LIN {X 0,Y 467.59,Z 100.362,A -85,B 0,C 180,E1 -7607.44,E2 -7607.44} C_VEL
LIN {X 0,Y 467.583,Z 100.361,A -85,B 0,C 180,E1 -7610.855,E2 -7610.855} C_VEL
LIN {X 0,Y 467.561,Z 100.367,A -85,B 0,C 180,E1 -7614.261,E2 -7614.261} C_VEL
LIN {X 0,Y 467.583,Z 100.359,A -85,B 0,C 180,E1 -7617.321,E2 -7617.321} C_VEL
LIN {X 0,Y 467.571,Z 100.367,A -85,B 0,C 180,E1 -7620.667,E2 -7620.667} C_VEL
LIN {X 0,Y 467.632,Z 100.488,A -85,B 0,C 180,E1 -7622.14,E2 -7622.14} C_VEL
LIN {X 0,Y 470.539,Z 113.37,A -85,B 0,C 180,E1 -7624.57,E2 -7624.57} C_VEL
LIN {X 0,Y 471.052,Z 117.501,A -85,B 0,C 180,E1 -7625.307,E2 -7625.307} C_VEL
LIN {X 0,Y 469.859,Z 138.203,A -85,B 0,C 180,E1 -7628.732,E2 -7628.732} C_VEL
LIN {X 0,Y 469.678,Z 141.309,A -85,B 0,C 180,E1 -7629.24,E2 -7629.24} C_VEL
LIN {X 0,Y 473.653,Z 162.605,A -85,B 0,C 180,E1 -7629.783,E2 -7629.783} C_VEL
LIN {X 0,Y 472.479,Z 278.914,A -85,B 0,C 180,E1 -7631.601,E2 -7631.601} C_VEL
LIN {X 0,Y 472.045,Z 293.392,A -85,B 0,C 180,E1 -7631.996,E2 -7631.996} C_VEL
LIN {X 0,Y 471.498,Z 306.65,A -85,B 0,C 180,E1 -7632.524,E2 -7632.524} C_VEL
LIN {X 0,Y 470.833,Z 320.055,A -85,B 0,C 180,E1 -7633.238,E2 -7633.238} C_VEL
LIN {X 0,Y 470.092,Z 333.562,A -85,B 0,C 180,E1 -7634.166,E2 -7634.166} C_VEL
LIN {X 0,Y 469.368,Z 345.002,A -85,B 0,C 180,E1 -7635.142,E2 -7635.142} C_VEL
LIN {X 0,Y 468.685,Z 356.491,A -85,B 0,C 180,E1 -7636.339,E2 -7636.339} C_VEL
LIN {X 0,Y 468.141,Z 365.96,A -85,B 0,C 180,E1 -7637.535,E2 -7637.535} C_VEL
LIN {X 0,Y 467.636,Z 375.295,A -85,B 0,C 180,E1 -7638.953,E2 -7638.953} C_VEL
LIN {X 0,Y 467.209,Z 383.442,A -85,B 0,C 180,E1 -7640.475,E2 -7640.475} C_VEL
LIN {X 0,Y 466.947,Z 389.181,A -85,B 0,C 180,E1 -7641.779,E2 -7641.779} C_VEL
LIN {X 0,Y 466.821,Z 393.865,A -85,B 0,C 180,E1 -7643.082,E2 -7643.082} C_VEL
LIN {X 0,Y 466.723,Z 398.729,A -85,B 0,C 180,E1 -7644.816,E2 -7644.816} C_VEL
LIN {X 0,Y 466.65,Z 402.107,A -85,B 0,C 180,E1 -7646.546,E2 -7646.546} C_VEL
LIN {X 0,Y 466.604,Z 404.094,A -85,B 0,C 180,E1 -7648.274,E2 -7648.274} C_VEL
LIN {X 0,Y 466.598,Z 404.732,A -85,B 0,C 180,E1 -7650,E2 -7650} C_VEL
LIN {X 0,Y 466.604,Z 404.034,A -85,B 0,C 180,E1 -7651.726,E2 -7651.726} C_VEL
LIN {X 0,Y 466.65,Z 401.99,A -85,B 0,C 180,E1 -7653.454,E2 -7653.454} C_VEL
LIN {X 0,Y 466.724,Z 398.543,A -85,B 0,C 180,E1 -7655.184,E2 -7655.184} C_VEL
LIN {X 0,Y 466.82,Z 393.586,A -85,B 0,C 180,E1 -7656.917,E2 -7656.917} C_VEL
LIN {X 0,Y 466.998,Z 386.974,A -85,B 0,C 180,E1 -7658.655,E2 -7658.655} C_VEL
LIN {X 0,Y 467.303,Z 379.612,A -85,B 0,C 180,E1 -7660.178,E2 -7660.178} C_VEL
LIN {X 0,Y 467.801,Z 370.456,A -85,B 0,C 180,E1 -7661.702,E2 -7661.702} C_VEL
LIN {X 0,Y 468.273,Z 360.859,A -85,B 0,C 180,E1 -7663.01,E2 -7663.01} C_VEL
LIN {X 0,Y 468.894,Z 350.221,A -85,B 0,C 180,E1 -7664.207,E2 -7664.207} C_VEL
LIN {X 0,Y 469.535,Z 338.457,A -85,B 0,C 180,E1 -7665.296,E2 -7665.296} C_VEL
LIN {X 0,Y 470.146,Z 326.953,A -85,B 0,C 180,E1 -7666.166,E2 -7666.166} C_VEL
LIN {X 0,Y 470.81,Z 314.697,A -85,B 0,C 180,E1 -7666.91,E2 -7666.91} C_VEL
LIN {X 0,Y 471.344,Z 300.603,A -85,B 0,C 180,E1 -7667.574,E2 -7667.574} C_VEL
LIN {X 0,Y 471.828,Z 287.015,A -85,B 0,C 180,E1 -7668.031,E2 -7668.031} C_VEL
LIN {X 0,Y 472.11,Z 273.417,A -85,B 0,C 180,E1 -7668.329,E2 -7668.329} C_VEL
LIN {X 0,Y 473.107,Z 162.279,A -85,B 0,C 180,E1 -7670.03,E2 -7670.03} C_VEL
LIN {X 0,Y 469.413,Z 141.425,A -85,B 0,C 180,E1 -7670.513,E2 -7670.513} C_VEL
LIN {X 0,Y 470.388,Z 121.167,A -85,B 0,C 180,E1 -7673.791,E2 -7673.791} C_VEL
LIN {X 0,Y 470.519,Z 114.09,A -85,B 0,C 180,E1 -7674.958,E2 -7674.958} C_VEL
LIN {X 0,Y 467.644,Z 100.358,A -85,B 0,C 180,E1 -7677.451,E2 -7677.451} C_VEL
LIN {X 0,Y 467.568,Z 100.367,A -85,B 0,C 180,E1 -7681.045,E2 -7681.045} C_VEL
LIN {X 0,Y 467.588,Z 100.368,A -85,B 0,C 180,E1 -7684.242,E2 -7684.242} C_VEL
LIN {X 0,Y 467.548,Z 100.366,A -85,B 0,C 180,E1 -7687.186,E2 -7687.186} C_VEL
LIN {X 0,Y 467.577,Z 100.366,A -85,B 0,C 180,E1 -7690.264,E2 -7690.264} C_VEL
LIN {X 0,Y 467.586,Z 100.362,A -85,B 0,C 180,E1 -7692.567,E2 -7692.567} C_VEL
LIN {X 0,Y 467.57,Z 100.364,A -85,B 0,C 180,E1 -7695.053,E2 -7695.053} C_VEL
LIN {X 0,Y 467.624,Z 100.361,A -85,B 0,C 180,E1 -7697.444,E2 -7697.444} C_VEL
LIN {X 0,Y 467.559,Z 100.365,A -85,B 0,C 180,E1 -7700.853,E2 -7700.853} C_VEL
LIN {X 0,Y 467.558,Z 100.365,A -85,B 0,C 180,E1 -7704.261,E2 -7704.261} C_VEL
LIN {X 0,Y 467.581,Z 100.369,A -85,B 0,C 180,E1 -7707.321,E2 -7707.321} C_VEL
LIN {X 0,Y 467.569,Z 100.364,A -85,B 0,C 180,E1 -7710.667,E2 -7710.667} C_VEL
LIN {X 0,Y 467.616,Z 100.366,A -85,B 0,C 180,E1 -7713.2,E2 -7713.2} C_VEL
LIN {X 0,Y 467.591,Z 100.362,A -85,B 0,C 180,E1 -7716.468,E2 -7716.468} C_VEL
LIN {X 0,Y 467.621,Z 100.357,A -85,B 0,C 180,E1 -7719.777,E2 -7719.777} C_VEL
LIN {X 0,Y 467.606,Z 100.362,A -85,B 0,C 180,E1 -7722.507,E2 -7722.507} C_VEL
LIN {X 0,Y 467.605,Z 100.362,A -85,B 0,C 180,E1 -7725.197,E2 -7725.197} C_VEL
LIN {X 0,Y 467.655,Z 100.353,A -85,B 0,C 180,E1 -7727.855,E2 -7727.855} C_VEL
LIN {X 0,Y 467.68,Z 100.35,A -85,B 0,C 180,E1 -7731.357,E2 -7731.357} C_VEL
LIN {X 0,Y 467.736,Z 100.344,A -85,B 0,C 180,E1 -7733.963,E2 -7733.963} C_VEL
LIN {X 0,Y 467.858,Z 100.327,A -85,B 0,C 180,E1 -7737.417,E2 -7737.417} C_VEL
LIN {X 0,Y 467.881,Z 100.328,A -85,B 0,C 180,E1 -7740,E2 -7740} C_VEL
LIN {X 0,Y 467.858,Z 100.331,A -85,B 0,C 180,E1 -7742.583,E2 -7742.583} C_VEL
LIN {X 0,Y 467.72,Z 100.352,A -85,B 0,C 180,E1 -7746.038,E2 -7746.038} C_VEL
LIN {X 0,Y 467.681,Z 100.35,A -85,B 0,C 180,E1 -7748.643,E2 -7748.643} C_VEL
LIN {X 0,Y 467.655,Z 100.357,A -85,B 0,C 180,E1 -7752.146,E2 -7752.146} C_VEL
LIN {X 0,Y 467.638,Z 100.361,A -85,B 0,C 180,E1 -7755.695,E2 -7755.695} C_VEL
LIN {X 0,Y 467.621,Z 100.36,A -85,B 0,C 180,E1 -7759.308,E2 -7759.308} C_VEL
LIN {X 0,Y 467.534,Z 100.37,A -85,B 0,C 180,E1 -7762.074,E2 -7762.074} C_VEL
LIN {X 0,Y 467.585,Z 100.363,A -85,B 0,C 180,E1 -7764.889,E2 -7764.889} C_VEL
LIN {X 0,Y 467.619,Z 100.36,A -85,B 0,C 180,E1 -7767.769,E2 -7767.769} C_VEL
LIN {X 0,Y 467.567,Z 100.368,A -85,B 0,C 180,E1 -7771.045,E2 -7771.045} C_VEL
LIN {X 0,Y 467.577,Z 100.362,A -85,B 0,C 180,E1 -7774.24,E2 -7774.24} C_VEL
LIN {X 0,Y 467.547,Z 100.372,A -85,B 0,C 180,E1 -7777.187,E2 -7777.187} C_VEL
LIN {X 0,Y 467.574,Z 100.363,A -85,B 0,C 180,E1 -7780.265,E2 -7780.265} C_VEL
LIN {X 0,Y 467.587,Z 100.365,A -85,B 0,C 180,E1 -7782.567,E2 -7782.567} C_VEL
LIN {X 0,Y 467.566,Z 100.368,A -85,B 0,C 180,E1 -7785.053,E2 -7785.053} C_VEL
LIN {X 0,Y 467.574,Z 100.369,A -85,B 0,C 180,E1 -7788.597,E2 -7788.597} C_VEL
LIN {X 0,Y 467.563,Z 100.365,A -85,B 0,C 180,E1 -7791.956,E2 -7791.956} C_VEL
LIN {X 0,Y 467.564,Z 100.365,A -85,B 0,C 180,E1 -7795.168,E2 -7795.168} C_VEL
LIN {X 0,Y 467.585,Z 100.368,A -85,B 0,C 180,E1 -7798.26,E2 -7798.26} C_VEL
LIN {X 0,Y 467.556,Z 100.365,A -85,B 0,C 180,E1 -7801.249,E2 -7801.249} C_VEL
LIN {X 0,Y 467.581,Z 100.369,A -85,B 0,C 180,E1 -7804.159,E2 -7804.159} C_VEL
LIN {X 0,Y 467.578,Z 100.362,A -85,B 0,C 180,E1 -7806.996,E2 -7806.996} C_VEL
LIN {X 0,Y 467.611,Z 100.363,A -85,B 0,C 180,E1 -7810.375,E2 -7810.375} C_VEL
LIN {X 0,Y 467.649,Z 100.469,A -85,B 0,C 180,E1 -7811.446,E2 -7811.446} C_VEL
LIN {X 0,Y 469.89,Z 112.337,A -85,B 0,C 180,E1 -7813.801,E2 -7813.801} C_VEL
LIN {X 0,Y 469.308,Z 114.722,A -85,B 0,C 180,E1 -7814.217,E2 -7814.217} C_VEL
LIN {X 0,Y 467.724,Z 117.234,A -85,B 0,C 180,E1 -7814.59,E2 -7814.59} C_VEL
LIN {X 0,Y 465.302,Z 120.97,A -85,B 0,C 180,E1 -7815.008,E2 -7815.008} C_VEL
LIN {X 0,Y 463.889,Z 124.864,A -85,B 0,C 180,E1 -7815.289,E2 -7815.289} C_VEL
LIN {X 0,Y 463.925,Z 127.986,A -85,B 0,C 180,E1 -7815.416,E2 -7815.416} C_VEL
LIN {X 0,Y 466.531,Z 140.838,A -85,B 0,C 180,E1 -7815.733,E2 -7815.733} C_VEL
LIN {X 0,Y 465.376,Z 258.301,A -85,B 0,C 180,E1 -7817.573,E2 -7817.573} C_VEL
LIN {X 0,Y 465.029,Z 272.977,A -85,B 0,C 180,E1 -7817.979,E2 -7817.979} C_VEL
LIN {X 0,Y 464.568,Z 286.896,A -85,B 0,C 180,E1 -7818.548,E2 -7818.548} C_VEL
LIN {X 0,Y 463.909,Z 300.717,A -85,B 0,C 180,E1 -7819.305,E2 -7819.305} C_VEL
LIN {X 0,Y 463.223,Z 313.085,A -85,B 0,C 180,E1 -7820.173,E2 -7820.173} C_VEL
LIN {X 0,Y 462.552,Z 325.536,A -85,B 0,C 180,E1 -7821.261,E2 -7821.261} C_VEL
LIN {X 0,Y 461.968,Z 335.732,A -85,B 0,C 180,E1 -7822.351,E2 -7822.351} C_VEL
LIN {X 0,Y 461.293,Z 345.908,A -85,B 0,C 180,E1 -7823.659,E2 -7823.659} C_VEL
LIN {X 0,Y 460.791,Z 354.325,A -85,B 0,C 180,E1 -7824.969,E2 -7824.969} C_VEL
LIN {X 0,Y 460.197,Z 362.395,A -85,B 0,C 180,E1 -7826.498,E2 -7826.498} C_VEL
LIN {X 0,Y 460.018,Z 368.058,A -85,B 0,C 180,E1 -7827.811,E2 -7827.811} C_VEL
LIN {X 0,Y 459.705,Z 372.702,A -85,B 0,C 180,E1 -7829.124,E2 -7829.124} C_VEL
LIN {X 0,Y 459.615,Z 377.518,A -85,B 0,C 180,E1 -7830.876,E2 -7830.876} C_VEL
LIN {X 0,Y 459.601,Z 380.867,A -85,B 0,C 180,E1 -7832.629,E2 -7832.629} C_VEL
LIN {X 0,Y 459.521,Z 382.844,A -85,B 0,C 180,E1 -7834.386,E2 -7834.386} C_VEL
LIN {X 0,Y 459.592,Z 383.48,A -85,B 0,C 180,E1 -7836.145,E2 -7836.145} C_VEL
LIN {X 0,Y 459.522,Z 382.783,A -85,B 0,C 180,E1 -7837.912,E2 -7837.912} C_VEL
LIN {X 0,Y 459.505,Z 380.734,A -85,B 0,C 180,E1 -7839.686,E2 -7839.686} C_VEL
LIN {X 0,Y 459.744,Z 377.272,A -85,B 0,C 180,E1 -7841.463,E2 -7841.463} C_VEL
LIN {X 0,Y 459.91,Z 372.284,A -85,B 0,C 180,E1 -7843.251,E2 -7843.251} C_VEL
LIN {X 0,Y 460.144,Z 367.43,A -85,B 0,C 180,E1 -7844.597,E2 -7844.597} C_VEL
LIN {X 0,Y 460.56,Z 360.387,A -85,B 0,C 180,E1 -7846.17,E2 -7846.17} C_VEL
LIN {X 0,Y 461.093,Z 351.616,A -85,B 0,C 180,E1 -7847.749,E2 -7847.749} C_VEL
LIN {X 0,Y 461.759,Z 341.549,A -85,B 0,C 180,E1 -7849.219,E2 -7849.219} C_VEL
LIN {X 0,Y 462.573,Z 330.076,A -85,B 0,C 180,E1 -7850.57,E2 -7850.57} C_VEL
LIN {X 0,Y 463.306,Z 318.29,A -85,B 0,C 180,E1 -7851.7,E2 -7851.7} C_VEL
LIN {X 0,Y 464.113,Z 305.504,A -85,B 0,C 180,E1 -7852.688,E2 -7852.688} C_VEL
LIN {X 0,Y 464.802,Z 292.175,A -85,B 0,C 180,E1 -7853.503,E2 -7853.503} C_VEL
LIN {X 0,Y 465.368,Z 278.873,A -85,B 0,C 180,E1 -7854.123,E2 -7854.123} C_VEL
LIN {X 0,Y 465.805,Z 265.448,A -85,B 0,C 180,E1 -7854.574,E2 -7854.574} C_VEL
LIN {X 0,Y 466.093,Z 250.619,A -85,B 0,C 180,E1 -7854.884,E2 -7854.884} C_VEL
LIN {X 0,Y 467.2,Z 140.6,A -85,B 0,C 180,E1 -7856.616,E2 -7856.616} C_VEL
LIN {X 0,Y 463.098,Z 122.09,A -85,B 0,C 180,E1 -7857.144,E2 -7857.144} C_VEL
LIN {X 0,Y 463.355,Z 115.546,A -85,B 0,C 180,E1 -7858.391,E2 -7858.391} C_VEL
LIN {X 0,Y 461.497,Z 105.781,A -85,B 0,C 180,E1 -7860.421,E2 -7860.421} C_VEL
LIN {X 0,Y 460.521,Z 101.248,A -85,B 0,C 180,E1 -7861.407,E2 -7861.407} C_VEL
LIN {X 0,Y 460.509,Z 101.246,A -85,B 0,C 180,E1 -7864.501,E2 -7864.501} C_VEL
LIN {X 0,Y 460.482,Z 101.25,A -85,B 0,C 180,E1 -7867.625,E2 -7867.625} C_VEL
LIN {X 0,Y 460.5,Z 101.247,A -85,B 0,C 180,E1 -7871.015,E2 -7871.015} C_VEL
LIN {X 0,Y 460.51,Z 101.244,A -85,B 0,C 180,E1 -7874.589,E2 -7874.589} C_VEL
LIN {X 0,Y 460.476,Z 101.252,A -85,B 0,C 180,E1 -7877.813,E2 -7877.813} C_VEL
LIN {X 0,Y 460.511,Z 101.236,A -85,B 0,C 180,E1 -7880.135,E2 -7880.135} C_VEL
LIN {X 0,Y 460.466,Z 101.252,A -85,B 0,C 180,E1 -7883.469,E2 -7883.469} C_VEL
LIN {X 0,Y 460.52,Z 101.244,A -85,B 0,C 180,E1 -7886.674,E2 -7886.674} C_VEL
LIN {X 0,Y 460.505,Z 101.242,A -85,B 0,C 180,E1 -7889.759,E2 -7889.759} C_VEL
LIN {X 0,Y 460.512,Z 101.249,A -85,B 0,C 180,E1 -7892.752,E2 -7892.752} C_VEL
LIN {X 0,Y 460.517,Z 101.243,A -85,B 0,C 180,E1 -7895.666,E2 -7895.666} C_VEL
LIN {X 0,Y 460.523,Z 101.243,A -85,B 0,C 180,E1 -7898.578,E2 -7898.578} C_VEL
LIN {X 0,Y 460.586,Z 101.23,A -85,B 0,C 180,E1 -7901.311,E2 -7901.311} C_VEL
LIN {X 0,Y 460.606,Z 101.234,A -85,B 0,C 180,E1 -7904.059,E2 -7904.059} C_VEL
LIN {X 0,Y 460.61,Z 101.23,A -85,B 0,C 180,E1 -7907.666,E2 -7907.666} C_VEL
LIN {X 0,Y 460.62,Z 101.223,A -85,B 0,C 180,E1 -7911.224,E2 -7911.224} C_VEL
LIN {X 0,Y 460.685,Z 101.226,A -85,B 0,C 180,E1 -7913.87,E2 -7913.87} C_VEL
LIN {X 0,Y 460.792,Z 101.206,A -85,B 0,C 180,E1 -7917.377,E2 -7917.377} C_VEL
LIN {X 0,Y 460.852,Z 101.203,A -85,B 0,C 180,E1 -7920,E2 -7920} C_VEL
LIN {X 0,Y 460.793,Z 101.208,A -85,B 0,C 180,E1 -7922.622,E2 -7922.622} C_VEL
LIN {X 0,Y 460.678,Z 101.22,A -85,B 0,C 180,E1 -7926.13,E2 -7926.13} C_VEL
LIN {X 0,Y 460.621,Z 101.23,A -85,B 0,C 180,E1 -7928.776,E2 -7928.776} C_VEL
LIN {X 0,Y 460.614,Z 101.228,A -85,B 0,C 180,E1 -7932.445,E2 -7932.445} C_VEL
LIN {X 0,Y 460.601,Z 101.226,A -85,B 0,C 180,E1 -7935.997,E2 -7935.997} C_VEL
LIN {X 0,Y 460.572,Z 101.238,A -85,B 0,C 180,E1 -7938.902,E2 -7938.902} C_VEL
LIN {X 0,Y 460.517,Z 101.244,A -85,B 0,C 180,E1 -7941.485,E2 -7941.485} C_VEL
LIN {X 0,Y 460.542,Z 101.237,A -85,B 0,C 180,E1 -7944.332,E2 -7944.332} C_VEL
LIN {X 0,Y 460.574,Z 101.238,A -85,B 0,C 180,E1 -7947.244,E2 -7947.244} C_VEL
LIN {X 0,Y 460.512,Z 101.243,A -85,B 0,C 180,E1 -7950.24,E2 -7950.24} C_VEL
LIN {X 0,Y 460.53,Z 101.243,A -85,B 0,C 180,E1 -7953.325,E2 -7953.325} C_VEL
LIN {X 0,Y 460.477,Z 101.252,A -85,B 0,C 180,E1 -7956.529,E2 -7956.529} C_VEL
LIN {X 0,Y 460.526,Z 101.234,A -85,B 0,C 180,E1 -7959.863,E2 -7959.863} C_VEL
LIN {X 0,Y 460.513,Z 101.244,A -85,B 0,C 180,E1 -7962.9,E2 -7962.9} C_VEL
LIN {X 0,Y 460.51,Z 101.243,A -85,B 0,C 180,E1 -7965.831,E2 -7965.831} C_VEL
LIN {X 0,Y 460.532,Z 101.241,A -85,B 0,C 180,E1 -7968.989,E2 -7968.989} C_VEL
LIN {X 0,Y 460.527,Z 101.24,A -85,B 0,C 180,E1 -7971.267,E2 -7971.267} C_VEL
LIN {X 0,Y 460.511,Z 101.243,A -85,B 0,C 180,E1 -7974.554,E2 -7974.554} C_VEL
LIN {X 0,Y 460.532,Z 101.24,A -85,B 0,C 180,E1 -7977.716,E2 -7977.716} C_VEL
LIN {X 0,Y 460.541,Z 101.243,A -85,B 0,C 180,E1 -7980.769,E2 -7980.769} C_VEL
LIN {X 0,Y 460.609,Z 101.434,A -85,B 0,C 180,E1 -7981.838,E2 -7981.838} C_VEL
LIN {X 0,Y 463.648,Z 114.783,A -85,B 0,C 180,E1 -7984.405,E2 -7984.405} C_VEL
LIN {X 0,Y 464.173,Z 119.706,A -85,B 0,C 180,E1 -7985.293,E2 -7985.293} C_VEL
LIN {X 0,Y 462.942,Z 139.583,A -85,B 0,C 180,E1 -7988.632,E2 -7988.632} C_VEL
LIN {X 0,Y 462.848,Z 141.135,A -85,B 0,C 180,E1 -7988.891,E2 -7988.891} C_VEL
LIN {X 0,Y 467.042,Z 163.344,A -85,B 0,C 180,E1 -7989.473,E2 -7989.473} C_VEL
LIN {X 0,Y 465.804,Z 278.587,A -85,B 0,C 180,E1 -7991.3,E2 -7991.3} C_VEL
LIN {X 0,Y 465.347,Z 293.36,A -85,B 0,C 180,E1 -7991.708,E2 -7991.708} C_VEL
LIN {X 0,Y 464.723,Z 307.37,A -85,B 0,C 180,E1 -7992.281,E2 -7992.281} C_VEL
LIN {X 0,Y 464.039,Z 320.484,A -85,B 0,C 180,E1 -7993,E2 -7993} C_VEL
LIN {X 0,Y 463.268,Z 333.695,A -85,B 0,C 180,E1 -7993.927,E2 -7993.927} C_VEL
LIN {X 0,Y 462.423,Z 346.25,A -85,B 0,C 180,E1 -7995.027,E2 -7995.027} C_VEL
LIN {X 0,Y 461.761,Z 356.524,A -85,B 0,C 180,E1 -7996.13,E2 -7996.13} C_VEL
LIN {X 0,Y 461.131,Z 366.58,A -85,B 0,C 180,E1 -7997.429,E2 -7997.429} C_VEL
LIN {X 0,Y 460.639,Z 375.254,A -85,B 0,C 180,E1 -7998.783,E2 -7998.783} C_VEL
LIN {X 0,Y 460.175,Z 383.372,A -85,B 0,C 180,E1 -8000.329,E2 -8000.329} C_VEL
LIN {X 0,Y 459.896,Z 389.099,A -85,B 0,C 180,E1 -8001.652,E2 -8001.652} C_VEL
LIN {X 0,Y 459.731,Z 393.764,A -85,B 0,C 180,E1 -8002.975,E2 -8002.975} C_VEL
LIN {X 0,Y 459.635,Z 398.612,A -85,B 0,C 180,E1 -8004.736,E2 -8004.736} C_VEL
LIN {X 0,Y 459.546,Z 401.974,A -85,B 0,C 180,E1 -8006.493,E2 -8006.493} C_VEL
LIN {X 0,Y 459.517,Z 403.944,A -85,B 0,C 180,E1 -8008.247,E2 -8008.247} C_VEL
LIN {X 0,Y 459.501,Z 404.567,A -85,B 0,C 180,E1 -8010,E2 -8010} C_VEL
LIN {X 0,Y 459.517,Z 403.855,A -85,B 0,C 180,E1 -8011.753,E2 -8011.753} C_VEL
LIN {X 0,Y 459.547,Z 401.796,A -85,B 0,C 180,E1 -8013.507,E2 -8013.507} C_VEL
LIN {X 0,Y 459.632,Z 398.333,A -85,B 0,C 180,E1 -8015.264,E2 -8015.264} C_VEL
LIN {X 0,Y 459.731,Z 393.359,A -85,B 0,C 180,E1 -8017.025,E2 -8017.025} C_VEL
LIN {X 0,Y 459.941,Z 386.728,A -85,B 0,C 180,E1 -8018.789,E2 -8018.789} C_VEL
LIN {X 0,Y 460.276,Z 379.344,A -85,B 0,C 180,E1 -8020.335,E2 -8020.335} C_VEL
LIN {X 0,Y 460.764,Z 370.149,A -85,B 0,C 180,E1 -8021.883,E2 -8021.883} C_VEL
LIN {X 0,Y 461.304,Z 360.521,A -85,B 0,C 180,E1 -8023.21,E2 -8023.21} C_VEL
LIN {X 0,Y 461.974,Z 349.845,A -85,B 0,C 180,E1 -8024.425,E2 -8024.425} C_VEL
LIN {X 0,Y 462.653,Z 338.031,A -85,B 0,C 180,E1 -8025.529,E2 -8025.529} C_VEL
LIN {X 0,Y 463.297,Z 326.464,A -85,B 0,C 180,E1 -8026.411,E2 -8026.411} C_VEL
LIN {X 0,Y 464.053,Z 313.041,A -85,B 0,C 180,E1 -8027.225,E2 -8027.225} C_VEL
LIN {X 0,Y 464.522,Z 299.889,A -85,B 0,C 180,E1 -8027.841,E2 -8027.841} C_VEL
LIN {X 0,Y 465.058,Z 286.076,A -85,B 0,C 180,E1 -8028.303,E2 -8028.303} C_VEL
LIN {X 0,Y 465.356,Z 271.908,A -85,B 0,C 180,E1 -8028.605,E2 -8028.605} C_VEL
LIN {X 0,Y 466.361,Z 163.164,A -85,B 0,C 180,E1 -8030.291,E2 -8030.291} C_VEL
LIN {X 0,Y 462.503,Z 141.199,A -85,B 0,C 180,E1 -8030.817,E2 -8030.817} C_VEL
LIN {X 0,Y 463.491,Z 122.252,A -85,B 0,C 180,E1 -8033.929,E2 -8033.929} C_VEL
LIN {X 0,Y 463.553,Z 115.172,A -85,B 0,C 180,E1 -8035.12,E2 -8035.12} C_VEL
LIN {X 0,Y 460.595,Z 101.236,A -85,B 0,C 180,E1 -8037.702,E2 -8037.702} C_VEL
LIN {X 0,Y 460.521,Z 101.245,A -85,B 0,C 180,E1 -8041.283,E2 -8041.283} C_VEL
LIN {X 0,Y 460.532,Z 101.243,A -85,B 0,C 180,E1 -8044.505,E2 -8044.505} C_VEL
LIN {X 0,Y 460.501,Z 101.246,A -85,B 0,C 180,E1 -8047.623,E2 -8047.623} C_VEL
LIN {X 0,Y 460.541,Z 101.242,A -85,B 0,C 180,E1 -8050.269,E2 -8050.269} C_VEL
LIN {X 0,Y 460.499,Z 101.246,A -85,B 0,C 180,E1 -8053.375,E2 -8053.375} C_VEL
LIN {X 0,Y 460.524,Z 101.241,A -85,B 0,C 180,E1 -8056.627,E2 -8056.627} C_VEL
LIN {X 0,Y 460.539,Z 101.246,A -85,B 0,C 180,E1 -8059.731,E2 -8059.731} C_VEL
LIN {X 0,Y 460.498,Z 101.244,A -85,B 0,C 180,E1 -8062.524,E2 -8062.524} C_VEL
LIN {X 0,Y 460.545,Z 101.244,A -85,B 0,C 180,E1 -8065.624,E2 -8065.624} C_VEL
LIN {X 0,Y 460.536,Z 101.241,A -85,B 0,C 180,E1 -8068.744,E2 -8068.744} C_VEL
LIN {X 0,Y 460.58,Z 101.234,A -85,B 0,C 180,E1 -8072.254,E2 -8072.254} C_VEL
LIN {X 0,Y 460.557,Z 101.239,A -85,B 0,C 180,E1 -8074.705,E2 -8074.705} C_VEL
LIN {X 0,Y 460.509,Z 101.244,A -85,B 0,C 180,E1 -8077.571,E2 -8077.571} C_VEL
LIN {X 0,Y 460.567,Z 101.237,A -85,B 0,C 180,E1 -8080.385,E2 -8080.385} C_VEL
LIN {X 0,Y 460.563,Z 101.24,A -85,B 0,C 180,E1 -8083.146,E2 -8083.146} C_VEL
LIN {X 0,Y 460.554,Z 101.237,A -85,B 0,C 180,E1 -8085.868,E2 -8085.868} C_VEL
LIN {X 0,Y 460.61,Z 101.236,A -85,B 0,C 180,E1 -8088.559,E2 -8088.559} C_VEL
LIN {X 0,Y 460.694,Z 101.222,A -85,B 0,C 180,E1 -8092.109,E2 -8092.109} C_VEL
LIN {X 0,Y 460.694,Z 101.224,A -85,B 0,C 180,E1 -8094.748,E2 -8094.748} C_VEL
LIN {X 0,Y 460.799,Z 101.207,A -85,B 0,C 180,E1 -8097.378,E2 -8097.378} C_VEL
LIN {X 0,Y 460.852,Z 101.204,A -85,B 0,C 180,E1 -8100,E2 -8100} C_VEL
LIN {X 0,Y 460.799,Z 101.209,A -85,B 0,C 180,E1 -8102.623,E2 -8102.623} C_VEL
LIN {X 0,Y 460.684,Z 101.229,A -85,B 0,C 180,E1 -8106.13,E2 -8106.13} C_VEL
LIN {X 0,Y 460.628,Z 101.228,A -85,B 0,C 180,E1 -8108.776,E2 -8108.776} C_VEL
LIN {X 0,Y 460.613,Z 101.231,A -85,B 0,C 180,E1 -8112.445,E2 -8112.445} C_VEL
LIN {X 0,Y 460.6,Z 101.236,A -85,B 0,C 180,E1 -8115.998,E2 -8115.998} C_VEL
LIN {X 0,Y 460.567,Z 101.243,A -85,B 0,C 180,E1 -8119.616,E2 -8119.616} C_VEL
LIN {X 0,Y 460.51,Z 101.243,A -85,B 0,C 180,E1 -8122.429,E2 -8122.429} C_VEL
LIN {X 0,Y 460.552,Z 101.241,A -85,B 0,C 180,E1 -8125.798,E2 -8125.798} C_VEL
LIN {X 0,Y 460.551,Z 101.238,A -85,B 0,C 180,E1 -8128.233,E2 -8128.233} C_VEL
LIN {X 0,Y 460.52,Z 101.249,A -85,B 0,C 180,E1 -8131.283,E2 -8131.283} C_VEL
LIN {X 0,Y 460.523,Z 101.242,A -85,B 0,C 180,E1 -8134.504,E2 -8134.504} C_VEL
LIN {X 0,Y 460.501,Z 101.245,A -85,B 0,C 180,E1 -8137.624,E2 -8137.624} C_VEL
LIN {X 0,Y 460.539,Z 101.24,A -85,B 0,C 180,E1 -8140.269,E2 -8140.269} C_VEL
LIN {X 0,Y 460.497,Z 101.246,A -85,B 0,C 180,E1 -8143.376,E2 -8143.376} C_VEL
LIN {X 0,Y 460.509,Z 101.249,A -85,B 0,C 180,E1 -8146.626,E2 -8146.626} C_VEL
LIN {X 0,Y 460.536,Z 101.239,A -85,B 0,C 180,E1 -8149.732,E2 -8149.732} C_VEL
LIN {X 0,Y 460.498,Z 101.252,A -85,B 0,C 180,E1 -8152.525,E2 -8152.525} C_VEL
LIN {X 0,Y 460.547,Z 101.238,A -85,B 0,C 180,E1 -8155.624,E2 -8155.624} C_VEL
LIN {X 0,Y 460.539,Z 101.242,A -85,B 0,C 180,E1 -8158.745,E2 -8158.745} C_VEL
LIN {X 0,Y 460.552,Z 101.245,A -85,B 0,C 180,E1 -8162.262,E2 -8162.262} C_VEL
LIN {X 0,Y 460.536,Z 101.241,A -85,B 0,C 180,E1 -8164.704,E2 -8164.704} C_VEL
LIN {X 0,Y 460.513,Z 101.244,A -85,B 0,C 180,E1 -8167.572,E2 -8167.572} C_VEL
LIN {X 0,Y 460.57,Z 101.242,A -85,B 0,C 180,E1 -8170.385,E2 -8170.385} C_VEL
LIN {X 0,Y 460.589,Z 101.323,A -85,B 0,C 180,E1 -8171.215,E2 -8171.215} C_VEL
LIN {X 0,Y 462.976,Z 113.738,A -85,B 0,C 180,E1 -8173.717,E2 -8173.717} C_VEL
LIN {X 0,Y 462.7,Z 122.021,A -85,B 0,C 180,E1 -8175.261,E2 -8175.261} C_VEL
LIN {X 0,Y 463.925,Z 127.986,A -85,B 0,C 180,E1 -8175.416,E2 -8175.416} C_VEL
LIN {X 0,Y 464.359,Z 133.792,A -85,B 0,C 180,E1 -8175.528,E2 -8175.528} C_VEL
LIN {X 0,Y 463.604,Z 139.673,A -85,B 0,C 180,E1 -8175.59,E2 -8175.59} C_VEL
LIN {X 0,Y 460.035,Z 155.401,A -85,B 0,C 180,E1 -8175.693,E2 -8175.693} C_VEL
LIN {X 0,Y 459.698,Z 159.403,A -85,B 0,C 180,E1 -8175.743,E2 -8175.743} C_VEL
LIN {X 0,Y 458.593,Z 259.062,A -85,B 0,C 180,E1 -8177.33,E2 -8177.33} C_VEL
LIN {X 0,Y 458.233,Z 273.507,A -85,B 0,C 180,E1 -8177.742,E2 -8177.742} C_VEL
LIN {X 0,Y 457.75,Z 287.335,A -85,B 0,C 180,E1 -8178.319,E2 -8178.319} C_VEL
LIN {X 0,Y 457.109,Z 300.226,A -85,B 0,C 180,E1 -8179.032,E2 -8179.032} C_VEL
LIN {X 0,Y 456.393,Z 312.723,A -85,B 0,C 180,E1 -8179.912,E2 -8179.912} C_VEL
LIN {X 0,Y 455.678,Z 325.021,A -85,B 0,C 180,E1 -8180.992,E2 -8180.992} C_VEL
LIN {X 0,Y 454.993,Z 336.5,A -85,B 0,C 180,E1 -8182.233,E2 -8182.233} C_VEL
LIN {X 0,Y 454.273,Z 346.547,A -85,B 0,C 180,E1 -8183.56,E2 -8183.56} C_VEL
LIN {X 0,Y 453.763,Z 354.889,A -85,B 0,C 180,E1 -8184.891,E2 -8184.891} C_VEL
LIN {X 0,Y 453.153,Z 362.879,A -85,B 0,C 180,E1 -8186.443,E2 -8186.443} C_VEL
LIN {X 0,Y 452.931,Z 368.508,A -85,B 0,C 180,E1 -8187.777,E2 -8187.777} C_VEL
LIN {X 0,Y 452.661,Z 374.429,A -85,B 0,C 180,E1 -8189.555,E2 -8189.555} C_VEL
LIN {X 0,Y 452.546,Z 377.853,A -85,B 0,C 180,E1 -8190.89,E2 -8190.89} C_VEL
LIN {X 0,Y 452.522,Z 381.145,A -85,B 0,C 180,E1 -8192.671,E2 -8192.671} C_VEL
LIN {X 0,Y 452.438,Z 383.057,A -85,B 0,C 180,E1 -8194.455,E2 -8194.455} C_VEL
LIN {X 0,Y 452.516,Z 383.623,A -85,B 0,C 180,E1 -8196.287,E2 -8196.287} C_VEL
LIN {X 0,Y 452.439,Z 382.881,A -85,B 0,C 180,E1 -8198.037,E2 -8198.037} C_VEL
LIN {X 0,Y 452.429,Z 380.778,A -85,B 0,C 180,E1 -8199.839,E2 -8199.839} C_VEL
LIN {X 0,Y 452.674,Z 377.262,A -85,B 0,C 180,E1 -8201.644,E2 -8201.644} C_VEL
LIN {X 0,Y 452.866,Z 372.216,A -85,B 0,C 180,E1 -8203.461,E2 -8203.461} C_VEL
LIN {X 0,Y 453.127,Z 367.299,A -85,B 0,C 180,E1 -8204.828,E2 -8204.828} C_VEL
LIN {X 0,Y 453.594,Z 360.188,A -85,B 0,C 180,E1 -8206.425,E2 -8206.425} C_VEL
LIN {X 0,Y 454.076,Z 352.712,A -85,B 0,C 180,E1 -8207.799,E2 -8207.799} C_VEL
LIN {X 0,Y 454.695,Z 343.678,A -85,B 0,C 180,E1 -8209.176,E2 -8209.176} C_VEL
LIN {X 0,Y 455.386,Z 334.686,A -85,B 0,C 180,E1 -8210.319,E2 -8210.319} C_VEL
LIN {X 0,Y 456.12,Z 323.897,A -85,B 0,C 180,E1 -8211.466,E2 -8211.466} C_VEL
LIN {X 0,Y 456.98,Z 311.373,A -85,B 0,C 180,E1 -8212.549,E2 -8212.549} C_VEL
LIN {X 0,Y 457.756,Z 298.993,A -85,B 0,C 180,E1 -8213.407,E2 -8213.407} C_VEL
LIN {X 0,Y 458.479,Z 285.304,A -85,B 0,C 180,E1 -8214.148,E2 -8214.148} C_VEL
LIN {X 0,Y 458.96,Z 271.706,A -85,B 0,C 180,E1 -8214.693,E2 -8214.693} C_VEL
LIN {X 0,Y 459.354,Z 257.984,A -85,B 0,C 180,E1 -8215.063,E2 -8215.063} C_VEL
LIN {X 0,Y 460.667,Z 141.91,A -85,B 0,C 180,E1 -8216.93,E2 -8216.93} C_VEL
LIN {X 0,Y 456.293,Z 122.254,A -85,B 0,C 180,E1 -8217.506,E2 -8217.506} C_VEL
LIN {X 0,Y 456.401,Z 116.481,A -85,B 0,C 180,E1 -8218.63,E2 -8218.63} C_VEL
LIN {X 0,Y 454.224,Z 105.584,A -85,B 0,C 180,E1 -8220.947,E2 -8220.947} C_VEL
LIN {X 0,Y 453.464,Z 102.128,A -85,B 0,C 180,E1 -8221.71,E2 -8221.71} C_VEL
LIN {X 0,Y 453.467,Z 102.122,A -85,B 0,C 180,E1 -8224.99,E2 -8224.99} C_VEL
LIN {X 0,Y 453.441,Z 102.128,A -85,B 0,C 180,E1 -8228.314,E2 -8228.314} C_VEL
LIN {X 0,Y 453.465,Z 102.123,A -85,B 0,C 180,E1 -8230.612,E2 -8230.612} C_VEL
LIN {X 0,Y 453.48,Z 102.12,A -85,B 0,C 180,E1 -8234.528,E2 -8234.528} C_VEL
LIN {X 0,Y 453.437,Z 102.127,A -85,B 0,C 180,E1 -8238.071,E2 -8238.071} C_VEL
LIN {X 0,Y 453.439,Z 102.117,A -85,B 0,C 180,E1 -8240.802,E2 -8240.802} C_VEL
LIN {X 0,Y 453.448,Z 102.122,A -85,B 0,C 180,E1 -8243.916,E2 -8243.916} C_VEL
LIN {X 0,Y 453.479,Z 102.123,A -85,B 0,C 180,E1 -8247.151,E2 -8247.151} C_VEL
LIN {X 0,Y 453.463,Z 102.119,A -85,B 0,C 180,E1 -8250.267,E2 -8250.267} C_VEL
LIN {X 0,Y 453.453,Z 102.122,A -85,B 0,C 180,E1 -8253.29,E2 -8253.29} C_VEL
LIN {X 0,Y 453.493,Z 102.119,A -85,B 0,C 180,E1 -8256.238,E2 -8256.238} C_VEL
LIN {X 0,Y 453.483,Z 102.122,A -85,B 0,C 180,E1 -8259.117,E2 -8259.117} C_VEL
LIN {X 0,Y 453.502,Z 102.113,A -85,B 0,C 180,E1 -8261.944,E2 -8261.944} C_VEL
LIN {X 0,Y 453.536,Z 102.115,A -85,B 0,C 180,E1 -8264.726,E2 -8264.726} C_VEL
LIN {X 0,Y 453.56,Z 102.115,A -85,B 0,C 180,E1 -8268.379,E2 -8268.379} C_VEL
LIN {X 0,Y 453.586,Z 102.1,A -85,B 0,C 180,E1 -8271.086,E2 -8271.086} C_VEL
LIN {X 0,Y 453.651,Z 102.101,A -85,B 0,C 180,E1 -8273.774,E2 -8273.774} C_VEL
LIN {X 0,Y 453.736,Z 102.085,A -85,B 0,C 180,E1 -8277.336,E2 -8277.336} C_VEL
LIN {X 0,Y 453.822,Z 102.078,A -85,B 0,C 180,E1 -8280,E2 -8280} C_VEL
LIN {X 0,Y 453.737,Z 102.086,A -85,B 0,C 180,E1 -8282.663,E2 -8282.663} C_VEL
LIN {X 0,Y 453.645,Z 102.095,A -85,B 0,C 180,E1 -8286.226,E2 -8286.226} C_VEL
LIN {X 0,Y 453.586,Z 102.107,A -85,B 0,C 180,E1 -8288.913,E2 -8288.913} C_VEL
LIN {X 0,Y 453.564,Z 102.106,A -85,B 0,C 180,E1 -8292.529,E2 -8292.529} C_VEL
LIN {X 0,Y 453.546,Z 102.104,A -85,B 0,C 180,E1 -8296.196,E2 -8296.196} C_VEL
LIN {X 0,Y 453.521,Z 102.118,A -85,B 0,C 180,E1 -8299.041,E2 -8299.041} C_VEL
LIN {X 0,Y 453.477,Z 102.118,A -85,B 0,C 180,E1 -8301.836,E2 -8301.836} C_VEL
LIN {X 0,Y 453.514,Z 102.116,A -85,B 0,C 180,E1 -8304.734,E2 -8304.734} C_VEL
LIN {X 0,Y 453.533,Z 102.111,A -85,B 0,C 180,E1 -8307.96,E2 -8307.96} C_VEL
LIN {X 0,Y 453.467,Z 102.12,A -85,B 0,C 180,E1 -8311.525,E2 -8311.525} C_VEL
LIN {X 0,Y 453.488,Z 102.121,A -85,B 0,C 180,E1 -8314.777,E2 -8314.777} C_VEL
LIN {X 0,Y 453.461,Z 102.124,A -85,B 0,C 180,E1 -8318.312,E2 -8318.312} C_VEL
LIN {X 0,Y 453.494,Z 102.115,A -85,B 0,C 180,E1 -8320.609,E2 -8320.609} C_VEL
LIN {X 0,Y 453.455,Z 102.121,A -85,B 0,C 180,E1 -8323.244,E2 -8323.244} C_VEL
LIN {X 0,Y 453.464,Z 102.12,A -85,B 0,C 180,E1 -8325.779,E2 -8325.779} C_VEL
LIN {X 0,Y 453.48,Z 102.126,A -85,B 0,C 180,E1 -8328.209,E2 -8328.209} C_VEL
LIN {X 0,Y 453.516,Z 102.114,A -85,B 0,C 180,E1 -8330.79,E2 -8330.79} C_VEL
LIN {X 0,Y 453.455,Z 102.124,A -85,B 0,C 180,E1 -8333.917,E2 -8333.917} C_VEL
LIN {X 0,Y 453.484,Z 102.114,A -85,B 0,C 180,E1 -8337.151,E2 -8337.151} C_VEL
LIN {X 0,Y 453.476,Z 102.123,A -85,B 0,C 180,E1 -8340.268,E2 -8340.268} C_VEL
LIN {X 0,Y 453.529,Z 102.186,A -85,B 0,C 180,E1 -8341.484,E2 -8341.484} C_VEL
LIN {X 0,Y 456.751,Z 116.2,A -85,B 0,C 180,E1 -8344.235,E2 -8344.235} C_VEL
LIN {X 0,Y 457.344,Z 120.581,A -85,B 0,C 180,E1 -8345.047,E2 -8345.047} C_VEL
LIN {X 0,Y 456.12,Z 139.593,A -85,B 0,C 180,E1 -8348.297,E2 -8348.297} C_VEL
LIN {X 0,Y 456.028,Z 140.975,A -85,B 0,C 180,E1 -8348.53,E2 -8348.53} C_VEL
LIN {X 0,Y 460.286,Z 163.129,A -85,B 0,C 180,E1 -8349.128,E2 -8349.128} C_VEL
LIN {X 0,Y 460.511,Z 170.27,A -85,B 0,C 180,E1 -8349.258,E2 -8349.258} C_VEL
LIN {X 0,Y 459.156,Z 278.322,A -85,B 0,C 180,E1 -8350.99,E2 -8350.99} C_VEL
LIN {X 0,Y 458.704,Z 292.376,A -85,B 0,C 180,E1 -8351.376,E2 -8351.376} C_VEL
LIN {X 0,Y 458.034,Z 306.598,A -85,B 0,C 180,E1 -8351.956,E2 -8351.956} C_VEL
LIN {X 0,Y 457.346,Z 319.532,A -85,B 0,C 180,E1 -8352.666,E2 -8352.666} C_VEL
LIN {X 0,Y 456.558,Z 332.427,A -85,B 0,C 180,E1 -8353.569,E2 -8353.569} C_VEL
LIN {X 0,Y 455.701,Z 344.002,A -85,B 0,C 180,E1 -8354.571,E2 -8354.571} C_VEL
LIN {X 0,Y 454.961,Z 354.623,A -85,B 0,C 180,E1 -8355.69,E2 -8355.69} C_VEL
LIN {X 0,Y 454.308,Z 364.585,A -85,B 0,C 180,E1 -8356.956,E2 -8356.956} C_VEL
LIN {X 0,Y 453.73,Z 373.891,A -85,B 0,C 180,E1 -8358.383,E2 -8358.383} C_VEL
LIN {X 0,Y 453.157,Z 382.271,A -85,B 0,C 180,E1 -8359.952,E2 -8359.952} C_VEL
LIN {X 0,Y 452.823,Z 389.023,A -85,B 0,C 180,E1 -8361.521,E2 -8361.521} C_VEL
LIN {X 0,Y 452.593,Z 395.033,A -85,B 0,C 180,E1 -8363.312,E2 -8363.312} C_VEL
LIN {X 0,Y 452.548,Z 398.499,A -85,B 0,C 180,E1 -8364.653,E2 -8364.653} C_VEL
LIN {X 0,Y 452.444,Z 401.844,A -85,B 0,C 180,E1 -8366.438,E2 -8366.438} C_VEL
LIN {X 0,Y 452.499,Z 402.992,A -85,B 0,C 180,E1 -8367.329,E2 -8367.329} C_VEL
LIN {X 0,Y 452.401,Z 404.265,A -85,B 0,C 180,E1 -8369.11,E2 -8369.11} C_VEL
LIN {X 0,Y 452.401,Z 404.203,A -85,B 0,C 180,E1 -8370.89,E2 -8370.89} C_VEL
LIN {X 0,Y 452.499,Z 402.808,A -85,B 0,C 180,E1 -8372.67,E2 -8372.67} C_VEL
LIN {X 0,Y 452.469,Z 400.039,A -85,B 0,C 180,E1 -8374.454,E2 -8374.454} C_VEL
LIN {X 0,Y 452.562,Z 395.819,A -85,B 0,C 180,E1 -8376.241,E2 -8376.241} C_VEL
LIN {X 0,Y 452.739,Z 390.019,A -85,B 0,C 180,E1 -8378.031,E2 -8378.031} C_VEL
LIN {X 0,Y 453.039,Z 383.478,A -85,B 0,C 180,E1 -8379.6,E2 -8379.6} C_VEL
LIN {X 0,Y 453.466,Z 375.353,A -85,B 0,C 180,E1 -8381.17,E2 -8381.17} C_VEL
LIN {X 0,Y 453.953,Z 366.835,A -85,B 0,C 180,E1 -8382.518,E2 -8382.518} C_VEL
LIN {X 0,Y 454.525,Z 356.54,A -85,B 0,C 180,E1 -8383.867,E2 -8383.867} C_VEL
LIN {X 0,Y 455.176,Z 346.179,A -85,B 0,C 180,E1 -8384.988,E2 -8384.988} C_VEL
LIN {X 0,Y 455.931,Z 334.934,A -85,B 0,C 180,E1 -8385.994,E2 -8385.994} C_VEL
LIN {X 0,Y 456.638,Z 322.659,A -85,B 0,C 180,E1 -8386.888,E2 -8386.888} C_VEL
LIN {X 0,Y 457.308,Z 309.815,A -85,B 0,C 180,E1 -8387.628,E2 -8387.628} C_VEL
LIN {X 0,Y 457.857,Z 295.417,A -85,B 0,C 180,E1 -8388.254,E2 -8388.254} C_VEL
LIN {X 0,Y 458.362,Z 281.589,A -85,B 0,C 180,E1 -8388.667,E2 -8388.667} C_VEL
LIN {X 0,Y 458.685,Z 261.118,A -85,B 0,C 180,E1 -8389.03,E2 -8389.03} C_VEL
LIN {X 0,Y 459.569,Z 163.868,A -85,B 0,C 180,E1 -8390.563,E2 -8390.563} C_VEL
LIN {X 0,Y 455.593,Z 141.106,A -85,B 0,C 180,E1 -8391.107,E2 -8391.107} C_VEL
LIN {X 0,Y 456.596,Z 123.328,A -85,B 0,C 180,E1 -8394.072,E2 -8394.072} C_VEL
LIN {X 0,Y 456.755,Z 117.344,A -85,B 0,C 180,E1 -8395.089,E2 -8395.089} C_VEL
LIN {X 0,Y 453.524,Z 102.118,A -85,B 0,C 180,E1 -8397.919,E2 -8397.919} C_VEL
LIN {X 0,Y 453.476,Z 102.124,A -85,B 0,C 180,E1 -8400.759,E2 -8400.759} C_VEL
LIN {X 0,Y 453.477,Z 102.123,A -85,B 0,C 180,E1 -8403.912,E2 -8403.912} C_VEL
LIN {X 0,Y 453.452,Z 102.122,A -85,B 0,C 180,E1 -8407.189,E2 -8407.189} C_VEL
LIN {X 0,Y 453.489,Z 102.119,A -85,B 0,C 180,E1 -8409.45,E2 -8409.45} C_VEL
LIN {X 0,Y 453.476,Z 102.126,A -85,B 0,C 180,E1 -8411.935,E2 -8411.935} C_VEL
LIN {X 0,Y 453.493,Z 102.12,A -85,B 0,C 180,E1 -8415.47,E2 -8415.47} C_VEL
LIN {X 0,Y 453.493,Z 102.119,A -85,B 0,C 180,E1 -8418.211,E2 -8418.211} C_VEL
LIN {X 0,Y 453.486,Z 102.118,A -85,B 0,C 180,E1 -8420.794,E2 -8420.794} C_VEL
LIN {X 0,Y 453.453,Z 102.124,A -85,B 0,C 180,E1 -8423.917,E2 -8423.917} C_VEL
LIN {X 0,Y 453.482,Z 102.123,A -85,B 0,C 180,E1 -8427.151,E2 -8427.151} C_VEL
LIN {X 0,Y 453.474,Z 102.119,A -85,B 0,C 180,E1 -8430.268,E2 -8430.268} C_VEL
LIN {X 0,Y 453.506,Z 102.122,A -85,B 0,C 180,E1 -8433.294,E2 -8433.294} C_VEL
LIN {X 0,Y 453.501,Z 102.116,A -85,B 0,C 180,E1 -8436.239,E2 -8436.239} C_VEL
LIN {X 0,Y 453.482,Z 102.124,A -85,B 0,C 180,E1 -8439.118,E2 -8439.118} C_VEL
LIN {X 0,Y 453.509,Z 102.115,A -85,B 0,C 180,E1 -8441.945,E2 -8441.945} C_VEL
LIN {X 0,Y 453.539,Z 102.118,A -85,B 0,C 180,E1 -8444.726,E2 -8444.726} C_VEL
LIN {X 0,Y 453.558,Z 102.112,A -85,B 0,C 180,E1 -8448.379,E2 -8448.379} C_VEL
LIN {X 0,Y 453.651,Z 102.098,A -85,B 0,C 180,E1 -8451.985,E2 -8451.985} C_VEL
LIN {X 0,Y 453.667,Z 102.1,A -85,B 0,C 180,E1 -8454.667,E2 -8454.667} C_VEL
LIN {X 0,Y 453.743,Z 102.086,A -85,B 0,C 180,E1 -8457.337,E2 -8457.337} C_VEL
LIN {X 0,Y 453.822,Z 102.08,A -85,B 0,C 180,E1 -8460,E2 -8460} C_VEL
LIN {X 0,Y 453.743,Z 102.088,A -85,B 0,C 180,E1 -8462.663,E2 -8462.663} C_VEL
LIN {X 0,Y 453.65,Z 102.103,A -85,B 0,C 180,E1 -8466.226,E2 -8466.226} C_VEL
LIN {X 0,Y 453.591,Z 102.104,A -85,B 0,C 180,E1 -8468.914,E2 -8468.914} C_VEL
LIN {X 0,Y 453.563,Z 102.109,A -85,B 0,C 180,E1 -8472.529,E2 -8472.529} C_VEL
LIN {X 0,Y 453.544,Z 102.113,A -85,B 0,C 180,E1 -8476.196,E2 -8476.196} C_VEL
LIN {X 0,Y 453.516,Z 102.115,A -85,B 0,C 180,E1 -8479.04,E2 -8479.04} C_VEL
LIN {X 0,Y 453.476,Z 102.123,A -85,B 0,C 180,E1 -8481.836,E2 -8481.836} C_VEL
LIN {X 0,Y 453.5,Z 102.116,A -85,B 0,C 180,E1 -8484.735,E2 -8484.735} C_VEL
LIN {X 0,Y 453.531,Z 102.113,A -85,B 0,C 180,E1 -8487.96,E2 -8487.96} C_VEL
LIN {X 0,Y 453.465,Z 102.125,A -85,B 0,C 180,E1 -8491.525,E2 -8491.525} C_VEL
LIN {X 0,Y 453.482,Z 102.121,A -85,B 0,C 180,E1 -8494.777,E2 -8494.777} C_VEL
LIN {X 0,Y 453.462,Z 102.121,A -85,B 0,C 180,E1 -8498.312,E2 -8498.312} C_VEL
LIN {X 0,Y 453.494,Z 102.12,A -85,B 0,C 180,E1 -8500.609,E2 -8500.609} C_VEL
LIN {X 0,Y 453.454,Z 102.125,A -85,B 0,C 180,E1 -8503.244,E2 -8503.244} C_VEL
LIN {X 0,Y 453.461,Z 102.121,A -85,B 0,C 180,E1 -8505.779,E2 -8505.779} C_VEL
LIN {X 0,Y 453.494,Z 102.117,A -85,B 0,C 180,E1 -8509.41,E2 -8509.41} C_VEL
LIN {X 0,Y 453.45,Z 102.126,A -85,B 0,C 180,E1 -8512.81,E2 -8512.81} C_VEL
LIN {X 0,Y 453.478,Z 102.122,A -85,B 0,C 180,E1 -8516.088,E2 -8516.088} C_VEL
LIN {X 0,Y 453.477,Z 102.119,A -85,B 0,C 180,E1 -8519.241,E2 -8519.241} C_VEL
LIN {X 0,Y 453.509,Z 102.122,A -85,B 0,C 180,E1 -8522.296,E2 -8522.296} C_VEL
LIN {X 0,Y 453.497,Z 102.116,A -85,B 0,C 180,E1 -8525.265,E2 -8525.265} C_VEL
LIN {X 0,Y 453.483,Z 102.123,A -85,B 0,C 180,E1 -8528.415,E2 -8528.415} C_VEL
LIN {X 0,Y 453.54,Z 102.207,A -85,B 0,C 180,E1 -8530.983,E2 -8530.983} C_VEL
LIN {X 0,Y 455.941,Z 114.355,A -85,B 0,C 180,E1 -8533.475,E2 -8533.475} C_VEL
LIN {X 0,Y 455.975,Z 118.935,A -85,B 0,C 180,E1 -8534.352,E2 -8534.352} C_VEL
LIN {X 0,Y 455.798,Z 122.197,A -85,B 0,C 180,E1 -8534.963,E2 -8534.963} C_VEL
LIN {X 0,Y 459.856,Z 143.11,A -85,B 0,C 180,E1 -8535.486,E2 -8535.486} C_VEL
LIN {X 0,Y 459.698,Z 159.403,A -85,B 0,C 180,E1 -8535.743,E2 -8535.743} C_VEL
LIN {X 0,Y 458.968,Z 165.248,A -85,B 0,C 180,E1 -8535.807,E2 -8535.807} C_VEL
LIN {X 0,Y 453.298,Z 184.251,A -85,B 0,C 180,E1 -8535.876,E2 -8535.876} C_VEL
LIN {X 0,Y 452.604,Z 190.094,A -85,B 0,C 180,E1 -8535.942,E2 -8535.942} C_VEL
LIN {X 0,Y 451.817,Z 259.721,A -85,B 0,C 180,E1 -8537.079,E2 -8537.079} C_VEL
LIN {X 0,Y 451.433,Z 274.007,A -85,B 0,C 180,E1 -8537.497,E2 -8537.497} C_VEL
LIN {X 0,Y 450.92,Z 287.753,A -85,B 0,C 180,E1 -8538.082,E2 -8538.082} C_VEL
LIN {X 0,Y 450.211,Z 301.464,A -85,B 0,C 180,E1 -8538.862,E2 -8538.862} C_VEL
LIN {X 0,Y 449.453,Z 313.758,A -85,B 0,C 180,E1 -8539.755,E2 -8539.755} C_VEL
LIN {X 0,Y 448.734,Z 325.932,A -85,B 0,C 180,E1 -8540.854,E2 -8540.854} C_VEL
LIN {X 0,Y 448.014,Z 337.224,A -85,B 0,C 180,E1 -8542.111,E2 -8542.111} C_VEL
LIN {X 0,Y 447.259,Z 347.17,A -85,B 0,C 180,E1 -8543.459,E2 -8543.459} C_VEL
LIN {X 0,Y 446.719,Z 355.436,A -85,B 0,C 180,E1 -8544.81,E2 -8544.81} C_VEL
LIN {X 0,Y 446.112,Z 363.355,A -85,B 0,C 180,E1 -8546.387,E2 -8546.387} C_VEL
LIN {X 0,Y 445.851,Z 368.934,A -85,B 0,C 180,E1 -8547.742,E2 -8547.742} C_VEL
LIN {X 0,Y 445.578,Z 374.787,A -85,B 0,C 180,E1 -8549.548,E2 -8549.548} C_VEL
LIN {X 0,Y 445.449,Z 378.184,A -85,B 0,C 180,E1 -8550.904,E2 -8550.904} C_VEL
LIN {X 0,Y 445.445,Z 381.409,A -85,B 0,C 180,E1 -8552.713,E2 -8552.713} C_VEL
LIN {X 0,Y 445.358,Z 383.258,A -85,B 0,C 180,E1 -8554.526,E2 -8554.526} C_VEL
LIN {X 0,Y 445.415,Z 383.781,A -85,B 0,C 180,E1 -8556.341,E2 -8556.341} C_VEL
LIN {X 0,Y 445.339,Z 382.98,A -85,B 0,C 180,E1 -8558.166,E2 -8558.166} C_VEL
LIN {X 0,Y 445.364,Z 380.826,A -85,B 0,C 180,E1 -8559.996,E2 -8559.996} C_VEL
LIN {X 0,Y 445.619,Z 377.255,A -85,B 0,C 180,E1 -8561.831,E2 -8561.831} C_VEL
LIN {X 0,Y 445.829,Z 372.152,A -85,B 0,C 180,E1 -8563.678,E2 -8563.678} C_VEL
LIN {X 0,Y 446.135,Z 367.175,A -85,B 0,C 180,E1 -8565.066,E2 -8565.066} C_VEL
LIN {X 0,Y 446.64,Z 359.998,A -85,B 0,C 180,E1 -8566.689,E2 -8566.689} C_VEL
LIN {X 0,Y 447.159,Z 352.447,A -85,B 0,C 180,E1 -8568.084,E2 -8568.084} C_VEL
LIN {X 0,Y 447.812,Z 343.736,A -85,B 0,C 180,E1 -8569.424,E2 -8569.424} C_VEL
LIN {X 0,Y 448.574,Z 334.236,A -85,B 0,C 180,E1 -8570.641,E2 -8570.641} C_VEL
LIN {X 0,Y 449.353,Z 323.324,A -85,B 0,C 180,E1 -8571.806,E2 -8571.806} C_VEL
LIN {X 0,Y 450.2,Z 311.913,A -85,B 0,C 180,E1 -8572.802,E2 -8572.802} C_VEL
LIN {X 0,Y 450.986,Z 299.854,A -85,B 0,C 180,E1 -8573.658,E2 -8573.658} C_VEL
LIN {X 0,Y 451.768,Z 286.37,A -85,B 0,C 180,E1 -8574.408,E2 -8574.408} C_VEL
LIN {X 0,Y 452.243,Z 273.136,A -85,B 0,C 180,E1 -8574.962,E2 -8574.962} C_VEL
LIN {X 0,Y 452.715,Z 258.966,A -85,B 0,C 180,E1 -8575.364,E2 -8575.364} C_VEL
LIN {X 0,Y 454.19,Z 143.33,A -85,B 0,C 180,E1 -8577.25,E2 -8577.25} C_VEL
LIN {X 0,Y 449.504,Z 122.412,A -85,B 0,C 180,E1 -8577.88,E2 -8577.88} C_VEL
LIN {X 0,Y 449.44,Z 117.448,A -85,B 0,C 180,E1 -8578.873,E2 -8578.873} C_VEL
LIN {X 0,Y 447.182,Z 106.533,A -85,B 0,C 180,E1 -8581.241,E2 -8581.241} C_VEL
LIN {X 0,Y 446.413,Z 103.007,A -85,B 0,C 180,E1 -8582.027,E2 -8582.027} C_VEL
LIN {X 0,Y 446.416,Z 103,A -85,B 0,C 180,E1 -8585.05,E2 -8585.05} C_VEL
LIN {X 0,Y 446.395,Z 103.007,A -85,B 0,C 180,E1 -8588.075,E2 -8588.075} C_VEL
LIN {X 0,Y 446.396,Z 103.007,A -85,B 0,C 180,E1 -8591.395,E2 -8591.395} C_VEL
LIN {X 0,Y 446.421,Z 103,A -85,B 0,C 180,E1 -8595.108,E2 -8595.108} C_VEL
LIN {X 0,Y 446.401,Z 103.002,A -85,B 0,C 180,E1 -8598.605,E2 -8598.605} C_VEL
LIN {X 0,Y 446.4,Z 103.003,A -85,B 0,C 180,E1 -8601.923,E2 -8601.923} C_VEL
LIN {X 0,Y 446.423,Z 103.003,A -85,B 0,C 180,E1 -8605.476,E2 -8605.476} C_VEL
LIN {X 0,Y 446.416,Z 103.002,A -85,B 0,C 180,E1 -8608.699,E2 -8608.699} C_VEL
LIN {X 0,Y 446.448,Z 102.996,A -85,B 0,C 180,E1 -8611.83,E2 -8611.83} C_VEL
LIN {X 0,Y 446.421,Z 103.002,A -85,B 0,C 180,E1 -8614.845,E2 -8614.845} C_VEL
LIN {X 0,Y 446.449,Z 102.992,A -85,B 0,C 180,E1 -8618.245,E2 -8618.245} C_VEL
LIN {X 0,Y 446.451,Z 102.99,A -85,B 0,C 180,E1 -8621.649,E2 -8621.649} C_VEL
LIN {X 0,Y 446.506,Z 102.994,A -85,B 0,C 180,E1 -8624.479,E2 -8624.479} C_VEL
LIN {X 0,Y 446.518,Z 102.99,A -85,B 0,C 180,E1 -8628.193,E2 -8628.193} C_VEL
LIN {X 0,Y 446.533,Z 102.979,A -85,B 0,C 180,E1 -8630.944,E2 -8630.944} C_VEL
LIN {X 0,Y 446.62,Z 102.976,A -85,B 0,C 180,E1 -8633.676,E2 -8633.676} C_VEL
LIN {X 0,Y 446.683,Z 102.963,A -85,B 0,C 180,E1 -8637.294,E2 -8637.294} C_VEL
LIN {X 0,Y 446.792,Z 102.954,A -85,B 0,C 180,E1 -8640,E2 -8640} C_VEL
LIN {X 0,Y 446.684,Z 102.965,A -85,B 0,C 180,E1 -8642.705,E2 -8642.705} C_VEL
LIN {X 0,Y 446.613,Z 102.97,A -85,B 0,C 180,E1 -8646.324,E2 -8646.324} C_VEL
LIN {X 0,Y 446.533,Z 102.986,A -85,B 0,C 180,E1 -8649.055,E2 -8649.055} C_VEL
LIN {X 0,Y 446.522,Z 102.984,A -85,B 0,C 180,E1 -8652.73,E2 -8652.73} C_VEL
LIN {X 0,Y 446.491,Z 102.983,A -85,B 0,C 180,E1 -8656.459,E2 -8656.459} C_VEL
LIN {X 0,Y 446.47,Z 102.995,A -85,B 0,C 180,E1 -8659.303,E2 -8659.303} C_VEL
LIN {X 0,Y 446.419,Z 102.997,A -85,B 0,C 180,E1 -8662.199,E2 -8662.199} C_VEL
LIN {X 0,Y 446.458,Z 102.994,A -85,B 0,C 180,E1 -8665.152,E2 -8665.152} C_VEL
LIN {X 0,Y 446.485,Z 102.989,A -85,B 0,C 180,E1 -8668.179,E2 -8668.179} C_VEL
LIN {X 0,Y 446.42,Z 102.997,A -85,B 0,C 180,E1 -8671.775,E2 -8671.775} C_VEL
LIN {X 0,Y 446.43,Z 103.003,A -85,B 0,C 180,E1 -8674.523,E2 -8674.523} C_VEL
LIN {X 0,Y 446.414,Z 103.002,A -85,B 0,C 180,E1 -8678.079,E2 -8678.079} C_VEL
LIN {X 0,Y 446.428,Z 102.999,A -85,B 0,C 180,E1 -8680.918,E2 -8680.918} C_VEL
LIN {X 0,Y 446.401,Z 103.001,A -85,B 0,C 180,E1 -8683.846,E2 -8683.846} C_VEL
LIN {X 0,Y 446.399,Z 103.007,A -85,B 0,C 180,E1 -8686.403,E2 -8686.403} C_VEL
LIN {X 0,Y 446.427,Z 102.998,A -85,B 0,C 180,E1 -8689.082,E2 -8689.082} C_VEL
LIN {X 0,Y 446.417,Z 103.003,A -85,B 0,C 180,E1 -8691.921,E2 -8691.921} C_VEL
LIN {X 0,Y 446.43,Z 102.997,A -85,B 0,C 180,E1 -8695.477,E2 -8695.477} C_VEL
LIN {X 0,Y 446.417,Z 102.999,A -85,B 0,C 180,E1 -8698.7,E2 -8698.7} C_VEL
LIN {X 0,Y 446.495,Z 103.068,A -85,B 0,C 180,E1 -8701.146,E2 -8701.146} C_VEL
LIN {X 0,Y 449.566,Z 116.449,A -85,B 0,C 180,E1 -8703.828,E2 -8703.828} C_VEL
LIN {X 0,Y 450.472,Z 121.559,A -85,B 0,C 180,E1 -8704.807,E2 -8704.807} C_VEL
LIN {X 0,Y 449.535,Z 135.742,A -85,B 0,C 180,E1 -8707.28,E2 -8707.28} C_VEL
LIN {X 0,Y 449.265,Z 141.095,A -85,B 0,C 180,E1 -8708.168,E2 -8708.168} C_VEL
LIN {X 0,Y 453.736,Z 164.113,A -85,B 0,C 180,E1 -8708.802,E2 -8708.802} C_VEL
LIN {X 0,Y 453.945,Z 171.881,A -85,B 0,C 180,E1 -8708.944,E2 -8708.944} C_VEL
LIN {X 0,Y 452.51,Z 279.317,A -85,B 0,C 180,E1 -8710.699,E2 -8710.699} C_VEL
LIN {X 0,Y 451.969,Z 293.7,A -85,B 0,C 180,E1 -8711.117,E2 -8711.117} C_VEL
LIN {X 0,Y 451.302,Z 306.968,A -85,B 0,C 180,E1 -8711.677,E2 -8711.677} C_VEL
LIN {X 0,Y 450.576,Z 320.006,A -85,B 0,C 180,E1 -8712.411,E2 -8712.411} C_VEL
LIN {X 0,Y 449.759,Z 332.599,A -85,B 0,C 180,E1 -8713.314,E2 -8713.314} C_VEL
LIN {X 0,Y 448.849,Z 344.111,A -85,B 0,C 180,E1 -8714.33,E2 -8714.33} C_VEL
LIN {X 0,Y 448.05,Z 354.684,A -85,B 0,C 180,E1 -8715.465,E2 -8715.465} C_VEL
LIN {X 0,Y 447.337,Z 364.918,A -85,B 0,C 180,E1 -8716.793,E2 -8716.793} C_VEL
LIN {X 0,Y 446.753,Z 373.878,A -85,B 0,C 180,E1 -8718.199,E2 -8718.199} C_VEL
LIN {X 0,Y 446.132,Z 382.228,A -85,B 0,C 180,E1 -8719.792,E2 -8719.792} C_VEL
LIN {X 0,Y 445.77,Z 388.952,A -85,B 0,C 180,E1 -8721.386,E2 -8721.386} C_VEL
LIN {X 0,Y 445.509,Z 394.933,A -85,B 0,C 180,E1 -8723.205,E2 -8723.205} C_VEL
LIN {X 0,Y 445.461,Z 398.391,A -85,B 0,C 180,E1 -8724.568,E2 -8724.568} C_VEL
LIN {X 0,Y 445.343,Z 401.716,A -85,B 0,C 180,E1 -8726.381,E2 -8726.381} C_VEL
LIN {X 0,Y 445.405,Z 402.853,A -85,B 0,C 180,E1 -8727.287,E2 -8727.287} C_VEL
LIN {X 0,Y 445.313,Z 404.106,A -85,B 0,C 180,E1 -8729.096,E2 -8729.096} C_VEL
LIN {X 0,Y 445.313,Z 404.028,A -85,B 0,C 180,E1 -8730.904,E2 -8730.904} C_VEL
LIN {X 0,Y 445.423,Z 402.617,A -85,B 0,C 180,E1 -8732.713,E2 -8732.713} C_VEL
LIN {X 0,Y 445.391,Z 399.83,A -85,B 0,C 180,E1 -8734.525,E2 -8734.525} C_VEL
LIN {X 0,Y 445.454,Z 395.59,A -85,B 0,C 180,E1 -8736.341,E2 -8736.341} C_VEL
LIN {X 0,Y 445.613,Z 391.396,A -85,B 0,C 180,E1 -8737.704,E2 -8737.704} C_VEL
LIN {X 0,Y 445.837,Z 386.214,A -85,B 0,C 180,E1 -8739.07,E2 -8739.07} C_VEL
LIN {X 0,Y 446.212,Z 378.772,A -85,B 0,C 180,E1 -8740.665,E2 -8740.665} C_VEL
LIN {X 0,Y 446.668,Z 370.972,A -85,B 0,C 180,E1 -8742.033,E2 -8742.033} C_VEL
LIN {X 0,Y 447.219,Z 361.761,A -85,B 0,C 180,E1 -8743.379,E2 -8743.379} C_VEL
LIN {X 0,Y 447.966,Z 351.197,A -85,B 0,C 180,E1 -8744.654,E2 -8744.654} C_VEL
LIN {X 0,Y 448.711,Z 339.724,A -85,B 0,C 180,E1 -8745.791,E2 -8745.791} C_VEL
LIN {X 0,Y 449.52,Z 327.014,A -85,B 0,C 180,E1 -8746.812,E2 -8746.812} C_VEL
LIN {X 0,Y 450.346,Z 313.4,A -85,B 0,C 180,E1 -8747.673,E2 -8747.673} C_VEL
LIN {X 0,Y 450.915,Z 299.672,A -85,B 0,C 180,E1 -8748.339,E2 -8748.339} C_VEL
LIN {X 0,Y 451.454,Z 285.89,A -85,B 0,C 180,E1 -8748.816,E2 -8748.816} C_VEL
LIN {X 0,Y 451.783,Z 271.838,A -85,B 0,C 180,E1 -8749.126,E2 -8749.126} C_VEL
LIN {X 0,Y 452.933,Z 165.174,A -85,B 0,C 180,E1 -8750.825,E2 -8750.825} C_VEL
LIN {X 0,Y 448.712,Z 140.828,A -85,B 0,C 180,E1 -8751.435,E2 -8751.435} C_VEL
LIN {X 0,Y 449.727,Z 122.983,A -85,B 0,C 180,E1 -8754.464,E2 -8754.464} C_VEL
LIN {X 0,Y 449.827,Z 118.744,A -85,B 0,C 180,E1 -8755.197,E2 -8755.197} C_VEL
LIN {X 0,Y 446.784,Z 104.394,A -85,B 0,C 180,E1 -8757.903,E2 -8757.903} C_VEL
LIN {X 0,Y 446.485,Z 102.996,A -85,B 0,C 180,E1 -8758.178,E2 -8758.178} C_VEL
LIN {X 0,Y 446.419,Z 103.004,A -85,B 0,C 180,E1 -8761.775,E2 -8761.775} C_VEL
LIN {X 0,Y 446.429,Z 103,A -85,B 0,C 180,E1 -8764.523,E2 -8764.523} C_VEL
LIN {X 0,Y 446.415,Z 103.005,A -85,B 0,C 180,E1 -8768.079,E2 -8768.079} C_VEL
LIN {X 0,Y 446.426,Z 102.997,A -85,B 0,C 180,E1 -8770.917,E2 -8770.917} C_VEL
LIN {X 0,Y 446.417,Z 103.006,A -85,B 0,C 180,E1 -8773.844,E2 -8773.844} C_VEL
LIN {X 0,Y 446.452,Z 102.995,A -85,B 0,C 180,E1 -8776.396,E2 -8776.396} C_VEL
LIN {X 0,Y 446.44,Z 103.001,A -85,B 0,C 180,E1 -8779.802,E2 -8779.802} C_VEL
LIN {X 0,Y 446.4,Z 103.004,A -85,B 0,C 180,E1 -8783.255,E2 -8783.255} C_VEL
LIN {X 0,Y 446.447,Z 102.995,A -85,B 0,C 180,E1 -8786.566,E2 -8786.566} C_VEL
LIN {X 0,Y 446.429,Z 102.997,A -85,B 0,C 180,E1 -8789.979,E2 -8789.979} C_VEL
LIN {X 0,Y 446.474,Z 102.994,A -85,B 0,C 180,E1 -8792.839,E2 -8792.839} C_VEL
LIN {X 0,Y 446.464,Z 102.993,A -85,B 0,C 180,E1 -8795.923,E2 -8795.923} C_VEL
LIN {X 0,Y 446.452,Z 102.998,A -85,B 0,C 180,E1 -8798.773,E2 -8798.773} C_VEL
LIN {X 0,Y 446.455,Z 102.994,A -85,B 0,C 180,E1 -8801.649,E2 -8801.649} C_VEL
LIN {X 0,Y 446.507,Z 102.99,A -85,B 0,C 180,E1 -8804.48,E2 -8804.48} C_VEL
LIN {X 0,Y 446.516,Z 102.988,A -85,B 0,C 180,E1 -8808.193,E2 -8808.193} C_VEL
LIN {X 0,Y 446.599,Z 102.976,A -85,B 0,C 180,E1 -8811.858,E2 -8811.858} C_VEL
LIN {X 0,Y 446.642,Z 102.977,A -85,B 0,C 180,E1 -8814.583,E2 -8814.583} C_VEL
LIN {X 0,Y 446.662,Z 102.973,A -85,B 0,C 180,E1 -8818.197,E2 -8818.197} C_VEL
LIN {X 0,Y 446.792,Z 102.955,A -85,B 0,C 180,E1 -8820,E2 -8820} C_VEL
LIN {X 0,Y 446.69,Z 102.966,A -85,B 0,C 180,E1 -8822.706,E2 -8822.706} C_VEL
LIN {X 0,Y 446.618,Z 102.978,A -85,B 0,C 180,E1 -8826.324,E2 -8826.324} C_VEL
LIN {X 0,Y 446.537,Z 102.983,A -85,B 0,C 180,E1 -8829.056,E2 -8829.056} C_VEL
LIN {X 0,Y 446.521,Z 102.985,A -85,B 0,C 180,E1 -8832.73,E2 -8832.73} C_VEL
LIN {X 0,Y 446.495,Z 102.991,A -85,B 0,C 180,E1 -8836.228,E2 -8836.228} C_VEL
LIN {X 0,Y 446.467,Z 102.995,A -85,B 0,C 180,E1 -8839.304,E2 -8839.304} C_VEL
LIN {X 0,Y 446.417,Z 102.999,A -85,B 0,C 180,E1 -8842.2,E2 -8842.2} C_VEL
LIN {X 0,Y 446.443,Z 102.998,A -85,B 0,C 180,E1 -8845.153,E2 -8845.153} C_VEL
LIN {X 0,Y 446.484,Z 102.99,A -85,B 0,C 180,E1 -8848.179,E2 -8848.179} C_VEL
LIN {X 0,Y 446.418,Z 103,A -85,B 0,C 180,E1 -8851.775,E2 -8851.775} C_VEL
LIN {X 0,Y 446.422,Z 102.998,A -85,B 0,C 180,E1 -8854.524,E2 -8854.524} C_VEL
LIN {X 0,Y 446.414,Z 102.999,A -85,B 0,C 180,E1 -8858.079,E2 -8858.079} C_VEL
LIN {X 0,Y 446.428,Z 103.004,A -85,B 0,C 180,E1 -8860.918,E2 -8860.918} C_VEL
LIN {X 0,Y 446.399,Z 103,A -85,B 0,C 180,E1 -8863.847,E2 -8863.847} C_VEL
LIN {X 0,Y 446.398,Z 103.004,A -85,B 0,C 180,E1 -8866.404,E2 -8866.404} C_VEL
LIN {X 0,Y 446.436,Z 102.996,A -85,B 0,C 180,E1 -8869.802,E2 -8869.802} C_VEL
LIN {X 0,Y 446.401,Z 103.001,A -85,B 0,C 180,E1 -8873.255,E2 -8873.255} C_VEL
LIN {X 0,Y 446.45,Z 103,A -85,B 0,C 180,E1 -8876.567,E2 -8876.567} C_VEL
LIN {X 0,Y 446.43,Z 103,A -85,B 0,C 180,E1 -8879.98,E2 -8879.98} C_VEL
LIN {X 0,Y 446.445,Z 102.996,A -85,B 0,C 180,E1 -8882.837,E2 -8882.837} C_VEL
LIN {X 0,Y 446.463,Z 102.997,A -85,B 0,C 180,E1 -8885.925,E2 -8885.925} C_VEL
LIN {X 0,Y 446.456,Z 102.997,A -85,B 0,C 180,E1 -8888.773,E2 -8888.773} C_VEL
LIN {X 0,Y 446.5,Z 103.021,A -85,B 0,C 180,E1 -8890.73,E2 -8890.73} C_VEL
LIN {X 0,Y 448.924,Z 115.21,A -85,B 0,C 180,E1 -8893.272,E2 -8893.272} C_VEL
LIN {X 0,Y 449.096,Z 119.459,A -85,B 0,C 180,E1 -8894.106,E2 -8894.106} C_VEL
LIN {X 0,Y 448.916,Z 122.37,A -85,B 0,C 180,E1 -8894.659,E2 -8894.659} C_VEL
LIN {X 0,Y 453.135,Z 143.719,A -85,B 0,C 180,E1 -8895.203,E2 -8895.203} C_VEL
LIN {X 0,Y 452.604,Z 190.094,A -85,B 0,C 180,E1 -8895.942,E2 -8895.942} C_VEL
LIN {X 0,Y 451.912,Z 195.941,A -85,B 0,C 180,E1 -8896.009,E2 -8896.009} C_VEL
LIN {X 0,Y 446.255,Z 214.959,A -85,B 0,C 180,E1 -8896.084,E2 -8896.084} C_VEL
LIN {X 0,Y 445.537,Z 220.807,A -85,B 0,C 180,E1 -8896.151,E2 -8896.151} C_VEL
LIN {X 0,Y 445.021,Z 260.346,A -85,B 0,C 180,E1 -8896.821,E2 -8896.821} C_VEL
LIN {X 0,Y 444.64,Z 274.476,A -85,B 0,C 180,E1 -8897.245,E2 -8897.245} C_VEL
LIN {X 0,Y 444.113,Z 288.144,A -85,B 0,C 180,E1 -8897.839,E2 -8897.839} C_VEL
LIN {X 0,Y 443.394,Z 300.94,A -85,B 0,C 180,E1 -8898.573,E2 -8898.573} C_VEL
LIN {X 0,Y 442.654,Z 313.362,A -85,B 0,C 180,E1 -8899.48,E2 -8899.48} C_VEL
LIN {X 0,Y 441.891,Z 325.507,A -85,B 0,C 180,E1 -8900.583,E2 -8900.583} C_VEL
LIN {X 0,Y 441.113,Z 336.097,A -85,B 0,C 180,E1 -8901.756,E2 -8901.756} C_VEL
LIN {X 0,Y 440.377,Z 346.301,A -85,B 0,C 180,E1 -8903.126,E2 -8903.126} C_VEL
LIN {X 0,Y 439.75,Z 354.742,A -85,B 0,C 180,E1 -8904.498,E2 -8904.498} C_VEL
LIN {X 0,Y 439.141,Z 362.828,A -85,B 0,C 180,E1 -8906.1,E2 -8906.1} C_VEL
LIN {X 0,Y 438.776,Z 369.345,A -85,B 0,C 180,E1 -8907.705,E2 -8907.705} C_VEL
LIN {X 0,Y 438.499,Z 375.142,A -85,B 0,C 180,E1 -8909.541,E2 -8909.541} C_VEL
LIN {X 0,Y 438.355,Z 378.503,A -85,B 0,C 180,E1 -8910.919,E2 -8910.919} C_VEL
LIN {X 0,Y 438.369,Z 381.659,A -85,B 0,C 180,E1 -8912.757,E2 -8912.757} C_VEL
LIN {X 0,Y 438.28,Z 383.458,A -85,B 0,C 180,E1 -8914.599,E2 -8914.599} C_VEL
LIN {X 0,Y 438.316,Z 383.932,A -85,B 0,C 180,E1 -8916.445,E2 -8916.445} C_VEL
LIN {X 0,Y 438.255,Z 383.081,A -85,B 0,C 180,E1 -8918.298,E2 -8918.298} C_VEL
LIN {X 0,Y 438.304,Z 380.876,A -85,B 0,C 180,E1 -8920.159,E2 -8920.159} C_VEL
LIN {X 0,Y 438.545,Z 377.253,A -85,B 0,C 180,E1 -8922.025,E2 -8922.025} C_VEL
LIN {X 0,Y 438.802,Z 372.094,A -85,B 0,C 180,E1 -8923.901,E2 -8923.901} C_VEL
LIN {X 0,Y 439.131,Z 367.056,A -85,B 0,C 180,E1 -8925.312,E2 -8925.312} C_VEL
LIN {X 0,Y 439.688,Z 359.814,A -85,B 0,C 180,E1 -8926.96,E2 -8926.96} C_VEL
LIN {X 0,Y 440.262,Z 352.191,A -85,B 0,C 180,E1 -8928.377,E2 -8928.377} C_VEL
LIN {X 0,Y 441,Z 342.997,A -85,B 0,C 180,E1 -8929.795,E2 -8929.795} C_VEL
LIN {X 0,Y 441.774,Z 333.797,A -85,B 0,C 180,E1 -8930.974,E2 -8930.974} C_VEL
LIN {X 0,Y 442.616,Z 322.765,A -85,B 0,C 180,E1 -8932.155,E2 -8932.155} C_VEL
LIN {X 0,Y 443.529,Z 311.203,A -85,B 0,C 180,E1 -8933.165,E2 -8933.165} C_VEL
LIN {X 0,Y 444.346,Z 298.934,A -85,B 0,C 180,E1 -8934.034,E2 -8934.034} C_VEL
LIN {X 0,Y 445.176,Z 285.122,A -85,B 0,C 180,E1 -8934.793,E2 -8934.793} C_VEL
LIN {X 0,Y 445.699,Z 272.343,A -85,B 0,C 180,E1 -8935.318,E2 -8935.318} C_VEL
LIN {X 0,Y 446.129,Z 258.253,A -85,B 0,C 180,E1 -8935.71,E2 -8935.71} C_VEL
LIN {X 0,Y 447.579,Z 143.926,A -85,B 0,C 180,E1 -8937.604,E2 -8937.604} C_VEL
LIN {X 0,Y 442.718,Z 122.565,A -85,B 0,C 180,E1 -8938.269,E2 -8938.269} C_VEL
LIN {X 0,Y 442.47,Z 118.446,A -85,B 0,C 180,E1 -8939.12,E2 -8939.12} C_VEL
LIN {X 0,Y 439.92,Z 106.273,A -85,B 0,C 180,E1 -8941.816,E2 -8941.816} C_VEL
LIN {X 0,Y 439.36,Z 103.884,A -85,B 0,C 180,E1 -8942.386,E2 -8942.386} C_VEL
LIN {X 0,Y 439.383,Z 103.878,A -85,B 0,C 180,E1 -8945.338,E2 -8945.338} C_VEL
LIN {X 0,Y 439.349,Z 103.882,A -85,B 0,C 180,E1 -8948.599,E2 -8948.599} C_VEL
LIN {X 0,Y 439.346,Z 103.883,A -85,B 0,C 180,E1 -8952.21,E2 -8952.21} C_VEL
LIN {X 0,Y 439.376,Z 103.875,A -85,B 0,C 180,E1 -8955.267,E2 -8955.267} C_VEL
LIN {X 0,Y 439.364,Z 103.879,A -85,B 0,C 180,E1 -8958.747,E2 -8958.747} C_VEL
LIN {X 0,Y 439.358,Z 103.881,A -85,B 0,C 180,E1 -8961.611,E2 -8961.611} C_VEL
LIN {X 0,Y 439.395,Z 103.875,A -85,B 0,C 180,E1 -8964.843,E2 -8964.843} C_VEL
LIN {X 0,Y 439.372,Z 103.877,A -85,B 0,C 180,E1 -8968.139,E2 -8968.139} C_VEL
LIN {X 0,Y 439.401,Z 103.875,A -85,B 0,C 180,E1 -8971.606,E2 -8971.606} C_VEL
LIN {X 0,Y 439.366,Z 103.876,A -85,B 0,C 180,E1 -8974.412,E2 -8974.412} C_VEL
LIN {X 0,Y 439.363,Z 103.874,A -85,B 0,C 180,E1 -8977.424,E2 -8977.424} C_VEL
LIN {X 0,Y 439.442,Z 103.871,A -85,B 0,C 180,E1 -8980.663,E2 -8980.663} C_VEL
LIN {X 0,Y 439.462,Z 103.869,A -85,B 0,C 180,E1 -8984.224,E2 -8984.224} C_VEL
LIN {X 0,Y 439.484,Z 103.864,A -85,B 0,C 180,E1 -8988.001,E2 -8988.001} C_VEL
LIN {X 0,Y 439.504,Z 103.855,A -85,B 0,C 180,E1 -8991.725,E2 -8991.725} C_VEL
LIN {X 0,Y 439.609,Z 103.848,A -85,B 0,C 180,E1 -8994.495,E2 -8994.495} C_VEL
LIN {X 0,Y 439.634,Z 103.85,A -85,B 0,C 180,E1 -8998.168,E2 -8998.168} C_VEL
LIN {X 0,Y 439.761,Z 103.829,A -85,B 0,C 180,E1 -9000,E2 -9000} C_VEL
LIN {X 0,Y 439.633,Z 103.843,A -85,B 0,C 180,E1 -9002.749,E2 -9002.749} C_VEL
LIN {X 0,Y 439.565,Z 103.847,A -85,B 0,C 180,E1 -9006.426,E2 -9006.426} C_VEL
LIN {X 0,Y 439.496,Z 103.864,A -85,B 0,C 180,E1 -9009.202,E2 -9009.202} C_VEL
LIN {X 0,Y 439.466,Z 103.864,A -85,B 0,C 180,E1 -9012.937,E2 -9012.937} C_VEL
LIN {X 0,Y 439.448,Z 103.86,A -85,B 0,C 180,E1 -9016.348,E2 -9016.348} C_VEL
LIN {X 0,Y 439.403,Z 103.871,A -85,B 0,C 180,E1 -9019.626,E2 -9019.626} C_VEL
LIN {X 0,Y 439.366,Z 103.877,A -85,B 0,C 180,E1 -9022.575,E2 -9022.575} C_VEL
LIN {X 0,Y 439.406,Z 103.872,A -85,B 0,C 180,E1 -9025.585,E2 -9025.585} C_VEL
LIN {X 0,Y 439.418,Z 103.872,A -85,B 0,C 180,E1 -9028.673,E2 -9028.673} C_VEL
LIN {X 0,Y 439.371,Z 103.876,A -85,B 0,C 180,E1 -9032.03,E2 -9032.03} C_VEL
LIN {X 0,Y 439.395,Z 103.872,A -85,B 0,C 180,E1 -9035.34,E2 -9035.34} C_VEL
LIN {X 0,Y 439.376,Z 103.873,A -85,B 0,C 180,E1 -9038.596,E2 -9038.596} C_VEL
LIN {X 0,Y 439.389,Z 103.874,A -85,B 0,C 180,E1 -9041.257,E2 -9041.257} C_VEL
LIN {X 0,Y 439.4,Z 103.869,A -85,B 0,C 180,E1 -9044.729,E2 -9044.729} C_VEL
LIN {X 0,Y 439.396,Z 103.877,A -85,B 0,C 180,E1 -9047.796,E2 -9047.796} C_VEL
LIN {X 0,Y 439.437,Z 103.873,A -85,B 0,C 180,E1 -9050.228,E2 -9050.228} C_VEL
LIN {X 0,Y 439.374,Z 103.879,A -85,B 0,C 180,E1 -9053.713,E2 -9053.713} C_VEL
LIN {X 0,Y 439.373,Z 103.871,A -85,B 0,C 180,E1 -9057.054,E2 -9057.054} C_VEL
LIN {X 0,Y 439.447,Z 104.013,A -85,B 0,C 180,E1 -9060.805,E2 -9060.805} C_VEL
LIN {X 0,Y 442.618,Z 117.678,A -85,B 0,C 180,E1 -9063.603,E2 -9063.603} C_VEL
LIN {X 0,Y 443.622,Z 123.161,A -85,B 0,C 180,E1 -9064.676,E2 -9064.676} C_VEL
LIN {X 0,Y 442.525,Z 138.518,A -85,B 0,C 180,E1 -9067.394,E2 -9067.394} C_VEL
LIN {X 0,Y 442.451,Z 140.962,A -85,B 0,C 180,E1 -9067.781,E2 -9067.781} C_VEL
LIN {X 0,Y 446.818,Z 163.01,A -85,B 0,C 180,E1 -9068.408,E2 -9068.408} C_VEL
LIN {X 0,Y 447.401,Z 167.617,A -85,B 0,C 180,E1 -9068.519,E2 -9068.519} C_VEL
LIN {X 0,Y 445.927,Z 277.965,A -85,B 0,C 180,E1 -9070.343,E2 -9070.343} C_VEL
LIN {X 0,Y 445.416,Z 292.026,A -85,B 0,C 180,E1 -9070.739,E2 -9070.739} C_VEL
LIN {X 0,Y 444.675,Z 306.244,A -85,B 0,C 180,E1 -9071.334,E2 -9071.334} C_VEL
LIN {X 0,Y 443.904,Z 319.363,A -85,B 0,C 180,E1 -9072.076,E2 -9072.076} C_VEL
LIN {X 0,Y 443.04,Z 331.366,A -85,B 0,C 180,E1 -9072.934,E2 -9072.934} C_VEL
LIN {X 0,Y 442.006,Z 344.234,A -85,B 0,C 180,E1 -9074.081,E2 -9074.081} C_VEL
LIN {X 0,Y 441.171,Z 354.755,A -85,B 0,C 180,E1 -9075.233,E2 -9075.233} C_VEL
LIN {X 0,Y 440.35,Z 365.547,A -85,B 0,C 180,E1 -9076.666,E2 -9076.666} C_VEL
LIN {X 0,Y 439.655,Z 375.175,A -85,B 0,C 180,E1 -9078.24,E2 -9078.24} C_VEL
LIN {X 0,Y 439.024,Z 383.209,A -85,B 0,C 180,E1 -9079.858,E2 -9079.858} C_VEL
LIN {X 0,Y 438.732,Z 388.885,A -85,B 0,C 180,E1 -9081.247,E2 -9081.247} C_VEL
LIN {X 0,Y 438.442,Z 394.839,A -85,B 0,C 180,E1 -9083.095,E2 -9083.095} C_VEL
LIN {X 0,Y 438.358,Z 398.287,A -85,B 0,C 180,E1 -9084.48,E2 -9084.48} C_VEL
LIN {X 0,Y 438.247,Z 401.589,A -85,B 0,C 180,E1 -9086.322,E2 -9086.322} C_VEL
LIN {X 0,Y 438.275,Z 403.498,A -85,B 0,C 180,E1 -9088.162,E2 -9088.162} C_VEL
LIN {X 0,Y 438.228,Z 404.066,A -85,B 0,C 180,E1 -9090,E2 -9090} C_VEL
LIN {X 0,Y 438.275,Z 403.306,A -85,B 0,C 180,E1 -9091.838,E2 -9091.838} C_VEL
LIN {X 0,Y 438.33,Z 402.423,A -85,B 0,C 180,E1 -9092.757,E2 -9092.757} C_VEL
LIN {X 0,Y 438.313,Z 399.618,A -85,B 0,C 180,E1 -9094.598,E2 -9094.598} C_VEL
LIN {X 0,Y 438.367,Z 395.357,A -85,B 0,C 180,E1 -9096.443,E2 -9096.443} C_VEL
LIN {X 0,Y 438.529,Z 391.141,A -85,B 0,C 180,E1 -9097.829,E2 -9097.829} C_VEL
LIN {X 0,Y 438.822,Z 384.957,A -85,B 0,C 180,E1 -9099.448,E2 -9099.448} C_VEL
LIN {X 0,Y 439.256,Z 377.23,A -85,B 0,C 180,E1 -9101.069,E2 -9101.069} C_VEL
LIN {X 0,Y 439.833,Z 368.241,A -85,B 0,C 180,E1 -9102.601,E2 -9102.601} C_VEL
LIN {X 0,Y 440.372,Z 359.424,A -85,B 0,C 180,E1 -9103.85,E2 -9103.85} C_VEL
LIN {X 0,Y 441.125,Z 348.615,A -85,B 0,C 180,E1 -9105.122,E2 -9105.122} C_VEL
LIN {X 0,Y 442,Z 336.643,A -85,B 0,C 180,E1 -9106.275,E2 -9106.275} C_VEL
LIN {X 0,Y 442.761,Z 324.868,A -85,B 0,C 180,E1 -9107.196,E2 -9107.196} C_VEL
LIN {X 0,Y 443.524,Z 311.861,A -85,B 0,C 180,E1 -9108.007,E2 -9108.007} C_VEL
LIN {X 0,Y 444.106,Z 298.861,A -85,B 0,C 180,E1 -9108.631,E2 -9108.631} C_VEL
LIN {X 0,Y 444.712,Z 284.762,A -85,B 0,C 180,E1 -9109.113,E2 -9109.113} C_VEL
LIN {X 0,Y 445.059,Z 269.898,A -85,B 0,C 180,E1 -9109.427,E2 -9109.427} C_VEL
LIN {X 0,Y 446.148,Z 165.773,A -85,B 0,C 180,E1 -9111.114,E2 -9111.114} C_VEL
LIN {X 0,Y 441.796,Z 140.756,A -85,B 0,C 180,E1 -9111.74,E2 -9111.74} C_VEL
LIN {X 0,Y 442.813,Z 124.138,A -85,B 0,C 180,E1 -9114.605,E2 -9114.605} C_VEL
LIN {X 0,Y 442.829,Z 119.798,A -85,B 0,C 180,E1 -9115.373,E2 -9115.373} C_VEL
LIN {X 0,Y 439.816,Z 105.697,A -85,B 0,C 180,E1 -9118.079,E2 -9118.079} C_VEL
LIN {X 0,Y 439.429,Z 103.873,A -85,B 0,C 180,E1 -9118.443,E2 -9118.443} C_VEL
LIN {X 0,Y 439.37,Z 103.884,A -85,B 0,C 180,E1 -9122.03,E2 -9122.03} C_VEL
LIN {X 0,Y 439.394,Z 103.873,A -85,B 0,C 180,E1 -9125.34,E2 -9125.34} C_VEL
LIN {X 0,Y 439.378,Z 103.876,A -85,B 0,C 180,E1 -9128.595,E2 -9128.595} C_VEL
LIN {X 0,Y 439.388,Z 103.875,A -85,B 0,C 180,E1 -9131.257,E2 -9131.257} C_VEL
LIN {X 0,Y 439.404,Z 103.872,A -85,B 0,C 180,E1 -9134.729,E2 -9134.729} C_VEL
LIN {X 0,Y 439.41,Z 103.877,A -85,B 0,C 180,E1 -9137.797,E2 -9137.797} C_VEL
LIN {X 0,Y 439.394,Z 103.874,A -85,B 0,C 180,E1 -9140.224,E2 -9140.224} C_VEL
LIN {X 0,Y 439.372,Z 103.881,A -85,B 0,C 180,E1 -9143.713,E2 -9143.713} C_VEL
LIN {X 0,Y 439.371,Z 103.879,A -85,B 0,C 180,E1 -9147.054,E2 -9147.054} C_VEL
LIN {X 0,Y 439.381,Z 103.875,A -85,B 0,C 180,E1 -9150.274,E2 -9150.274} C_VEL
LIN {X 0,Y 439.427,Z 103.874,A -85,B 0,C 180,E1 -9153.396,E2 -9153.396} C_VEL
LIN {X 0,Y 439.385,Z 103.875,A -85,B 0,C 180,E1 -9156.43,E2 -9156.43} C_VEL
LIN {X 0,Y 439.387,Z 103.877,A -85,B 0,C 180,E1 -9159.397,E2 -9159.397} C_VEL
LIN {X 0,Y 439.429,Z 103.87,A -85,B 0,C 180,E1 -9162.31,E2 -9162.31} C_VEL
LIN {X 0,Y 439.446,Z 103.87,A -85,B 0,C 180,E1 -9165.174,E2 -9165.174} C_VEL
LIN {X 0,Y 439.482,Z 103.863,A -85,B 0,C 180,E1 -9168.001,E2 -9168.001} C_VEL
LIN {X 0,Y 439.547,Z 103.854,A -85,B 0,C 180,E1 -9171.726,E2 -9171.726} C_VEL
LIN {X 0,Y 439.617,Z 103.853,A -85,B 0,C 180,E1 -9174.496,E2 -9174.496} C_VEL
LIN {X 0,Y 439.632,Z 103.848,A -85,B 0,C 180,E1 -9178.168,E2 -9178.168} C_VEL
LIN {X 0,Y 439.761,Z 103.831,A -85,B 0,C 180,E1 -9180,E2 -9180} C_VEL
LIN {X 0,Y 439.64,Z 103.844,A -85,B 0,C 180,E1 -9182.749,E2 -9182.749} C_VEL
LIN {X 0,Y 439.59,Z 103.852,A -85,B 0,C 180,E1 -9186.426,E2 -9186.426} C_VEL
LIN {X 0,Y 439.499,Z 103.86,A -85,B 0,C 180,E1 -9189.202,E2 -9189.202} C_VEL
LIN {X 0,Y 439.465,Z 103.864,A -85,B 0,C 180,E1 -9192.938,E2 -9192.938} C_VEL
LIN {X 0,Y 439.445,Z 103.868,A -85,B 0,C 180,E1 -9196.348,E2 -9196.348} C_VEL
LIN {X 0,Y 439.401,Z 103.879,A -85,B 0,C 180,E1 -9199.627,E2 -9199.627} C_VEL
LIN {X 0,Y 439.363,Z 103.877,A -85,B 0,C 180,E1 -9202.576,E2 -9202.576} C_VEL
LIN {X 0,Y 439.398,Z 103.879,A -85,B 0,C 180,E1 -9205.586,E2 -9205.586} C_VEL
LIN {X 0,Y 439.417,Z 103.871,A -85,B 0,C 180,E1 -9208.674,E2 -9208.674} C_VEL
LIN {X 0,Y 439.368,Z 103.877,A -85,B 0,C 180,E1 -9212.03,E2 -9212.03} C_VEL
LIN {X 0,Y 439.392,Z 103.878,A -85,B 0,C 180,E1 -9215.34,E2 -9215.34} C_VEL
LIN {X 0,Y 439.377,Z 103.878,A -85,B 0,C 180,E1 -9218.596,E2 -9218.596} C_VEL
LIN {X 0,Y 439.389,Z 103.877,A -85,B 0,C 180,E1 -9221.257,E2 -9221.257} C_VEL
LIN {X 0,Y 439.399,Z 103.879,A -85,B 0,C 180,E1 -9224.73,E2 -9224.73} C_VEL
LIN {X 0,Y 439.385,Z 103.874,A -85,B 0,C 180,E1 -9227.795,E2 -9227.795} C_VEL
LIN {X 0,Y 439.389,Z 103.876,A -85,B 0,C 180,E1 -9230.224,E2 -9230.224} C_VEL
LIN {X 0,Y 439.373,Z 103.876,A -85,B 0,C 180,E1 -9233.713,E2 -9233.713} C_VEL
LIN {X 0,Y 439.374,Z 103.877,A -85,B 0,C 180,E1 -9237.054,E2 -9237.054} C_VEL
LIN {X 0,Y 439.379,Z 103.882,A -85,B 0,C 180,E1 -9240.274,E2 -9240.274} C_VEL
LIN {X 0,Y 439.382,Z 103.875,A -85,B 0,C 180,E1 -9243.393,E2 -9243.393} C_VEL
LIN {X 0,Y 439.385,Z 103.878,A -85,B 0,C 180,E1 -9246.43,E2 -9246.43} C_VEL
LIN {X 0,Y 439.391,Z 103.878,A -85,B 0,C 180,E1 -9249.397,E2 -9249.397} C_VEL
LIN {X 0,Y 439.439,Z 103.997,A -85,B 0,C 180,E1 -9250.502,E2 -9250.502} C_VEL
LIN {X 0,Y 441.731,Z 115.424,A -85,B 0,C 180,E1 -9252.927,E2 -9252.927} C_VEL
LIN {X 0,Y 442.232,Z 119.979,A -85,B 0,C 180,E1 -9253.853,E2 -9253.853} C_VEL
LIN {X 0,Y 442.083,Z 122.754,A -85,B 0,C 180,E1 -9254.349,E2 -9254.349} C_VEL
LIN {X 0,Y 446.434,Z 144.437,A -85,B 0,C 180,E1 -9254.915,E2 -9254.915} C_VEL
LIN {X 0,Y 445.537,Z 220.807,A -85,B 0,C 180,E1 -9256.151,E2 -9256.151} C_VEL
LIN {X 0,Y 444.806,Z 226.656,A -85,B 0,C 180,E1 -9256.217,E2 -9256.217} C_VEL
LIN {X 0,Y 439.093,Z 245.659,A -85,B 0,C 180,E1 -9256.294,E2 -9256.294} C_VEL
LIN {X 0,Y 438.449,Z 251.503,A -85,B 0,C 180,E1 -9256.365,E2 -9256.365} C_VEL
LIN {X 0,Y 438.171,Z 266.376,A -85,B 0,C 180,E1 -9256.699,E2 -9256.699} C_VEL
LIN {X 0,Y 437.727,Z 279.985,A -85,B 0,C 180,E1 -9257.187,E2 -9257.187} C_VEL
LIN {X 0,Y 437.109,Z 292.826,A -85,B 0,C 180,E1 -9257.818,E2 -9257.818} C_VEL
LIN {X 0,Y 436.324,Z 305.464,A -85,B 0,C 180,E1 -9258.62,E2 -9258.62} C_VEL
LIN {X 0,Y 435.459,Z 318.326,A -85,B 0,C 180,E1 -9259.657,E2 -9259.657} C_VEL
LIN {X 0,Y 434.616,Z 329.903,A -85,B 0,C 180,E1 -9260.812,E2 -9260.812} C_VEL
LIN {X 0,Y 433.938,Z 340.378,A -85,B 0,C 180,E1 -9262.087,E2 -9262.087} C_VEL
LIN {X 0,Y 433.141,Z 349.858,A -85,B 0,C 180,E1 -9263.478,E2 -9263.478} C_VEL
LIN {X 0,Y 432.436,Z 358.94,A -85,B 0,C 180,E1 -9265.106,E2 -9265.106} C_VEL
LIN {X 0,Y 431.902,Z 366.253,A -85,B 0,C 180,E1 -9266.735,E2 -9266.735} C_VEL
LIN {X 0,Y 431.533,Z 372.824,A -85,B 0,C 180,E1 -9268.6,E2 -9268.6} C_VEL
LIN {X 0,Y 431.345,Z 377.776,A -85,B 0,C 180,E1 -9270.467,E2 -9270.467} C_VEL
LIN {X 0,Y 431.251,Z 380.531,A -85,B 0,C 180,E1 -9271.868,E2 -9271.868} C_VEL
LIN {X 0,Y 431.276,Z 381.908,A -85,B 0,C 180,E1 -9272.802,E2 -9272.802} C_VEL
LIN {X 0,Y 431.203,Z 383.658,A -85,B 0,C 180,E1 -9274.675,E2 -9274.675} C_VEL
LIN {X 0,Y 431.214,Z 384.083,A -85,B 0,C 180,E1 -9276.551,E2 -9276.551} C_VEL
LIN {X 0,Y 431.154,Z 383.183,A -85,B 0,C 180,E1 -9278.436,E2 -9278.436} C_VEL
LIN {X 0,Y 431.25,Z 380.928,A -85,B 0,C 180,E1 -9280.327,E2 -9280.327} C_VEL
LIN {X 0,Y 431.505,Z 377.199,A -85,B 0,C 180,E1 -9282.248,E2 -9282.248} C_VEL
LIN {X 0,Y 431.764,Z 372.038,A -85,B 0,C 180,E1 -9284.132,E2 -9284.132} C_VEL
LIN {X 0,Y 432.123,Z 366.942,A -85,B 0,C 180,E1 -9285.566,E2 -9285.566} C_VEL
LIN {X 0,Y 432.731,Z 359.636,A -85,B 0,C 180,E1 -9287.242,E2 -9287.242} C_VEL
LIN {X 0,Y 433.35,Z 351.941,A -85,B 0,C 180,E1 -9288.681,E2 -9288.681} C_VEL
LIN {X 0,Y 434.246,Z 342.332,A -85,B 0,C 180,E1 -9290.166,E2 -9290.166} C_VEL
LIN {X 0,Y 435.143,Z 331.316,A -85,B 0,C 180,E1 -9291.558,E2 -9291.558} C_VEL
LIN {X 0,Y 436.124,Z 319.674,A -85,B 0,C 180,E1 -9292.753,E2 -9292.753} C_VEL
LIN {X 0,Y 437.146,Z 306.71,A -85,B 0,C 180,E1 -9293.824,E2 -9293.824} C_VEL
LIN {X 0,Y 438.024,Z 294.002,A -85,B 0,C 180,E1 -9294.656,E2 -9294.656} C_VEL
LIN {X 0,Y 438.709,Z 281.078,A -85,B 0,C 180,E1 -9295.311,E2 -9295.311} C_VEL
LIN {X 0,Y 439.274,Z 267.489,A -85,B 0,C 180,E1 -9295.812,E2 -9295.812} C_VEL
LIN {X 0,Y 439.633,Z 253.505,A -85,B 0,C 180,E1 -9296.146,E2 -9296.146} C_VEL
LIN {X 0,Y 441.054,Z 144.955,A -85,B 0,C 180,E1 -9297.957,E2 -9297.957} C_VEL
LIN {X 0,Y 436.318,Z 124.535,A -85,B 0,C 180,E1 -9298.597,E2 -9298.597} C_VEL
LIN {X 0,Y 435.894,Z 122.723,A -85,B 0,C 180,E1 -9298.675,E2 -9298.675} C_VEL
LIN {X 0,Y 434.525,Z 114.48,A -85,B 0,C 180,E1 -9300.479,E2 -9300.479} C_VEL
LIN {X 0,Y 432.313,Z 104.759,A -85,B 0,C 180,E1 -9302.72,E2 -9302.72} C_VEL
LIN {X 0,Y 432.332,Z 104.761,A -85,B 0,C 180,E1 -9305.818,E2 -9305.818} C_VEL
LIN {X 0,Y 432.313,Z 104.758,A -85,B 0,C 180,E1 -9308.709,E2 -9308.709} C_VEL
LIN {X 0,Y 432.301,Z 104.763,A -85,B 0,C 180,E1 -9311.801,E2 -9311.801} C_VEL
LIN {X 0,Y 432.333,Z 104.755,A -85,B 0,C 180,E1 -9314.348,E2 -9314.348} C_VEL
LIN {X 0,Y 432.303,Z 104.757,A -85,B 0,C 180,E1 -9317.018,E2 -9317.018} C_VEL
LIN {X 0,Y 432.289,Z 104.75,A -85,B 0,C 180,E1 -9319.828,E2 -9319.828} C_VEL
LIN {X 0,Y 432.3,Z 104.762,A -85,B 0,C 180,E1 -9323.021,E2 -9323.021} C_VEL
LIN {X 0,Y 432.334,Z 104.754,A -85,B 0,C 180,E1 -9326.002,E2 -9326.002} C_VEL
LIN {X 0,Y 432.347,Z 104.751,A -85,B 0,C 180,E1 -9329.49,E2 -9329.49} C_VEL
LIN {X 0,Y 432.339,Z 104.754,A -85,B 0,C 180,E1 -9331.873,E2 -9331.873} C_VEL
LIN {X 0,Y 432.322,Z 104.76,A -85,B 0,C 180,E1 -9334.997,E2 -9334.997} C_VEL
LIN {X 0,Y 432.358,Z 104.746,A -85,B 0,C 180,E1 -9338.045,E2 -9338.045} C_VEL
LIN {X 0,Y 432.385,Z 104.745,A -85,B 0,C 180,E1 -9341.029,E2 -9341.029} C_VEL
LIN {X 0,Y 432.43,Z 104.743,A -85,B 0,C 180,E1 -9343.961,E2 -9343.961} C_VEL
LIN {X 0,Y 432.46,Z 104.737,A -85,B 0,C 180,E1 -9347.803,E2 -9347.803} C_VEL
LIN {X 0,Y 432.465,Z 104.731,A -85,B 0,C 180,E1 -9351.59,E2 -9351.59} C_VEL
LIN {X 0,Y 432.585,Z 104.724,A -85,B 0,C 180,E1 -9354.406,E2 -9354.406} C_VEL
LIN {X 0,Y 432.604,Z 104.726,A -85,B 0,C 180,E1 -9358.138,E2 -9358.138} C_VEL
LIN {X 0,Y 432.731,Z 104.705,A -85,B 0,C 180,E1 -9360,E2 -9360} C_VEL
LIN {X 0,Y 432.585,Z 104.721,A -85,B 0,C 180,E1 -9362.794,E2 -9362.794} C_VEL
LIN {X 0,Y 432.58,Z 104.723,A -85,B 0,C 180,E1 -9365.594,E2 -9365.594} C_VEL
LIN {X 0,Y 432.464,Z 104.738,A -85,B 0,C 180,E1 -9368.41,E2 -9368.41} C_VEL
LIN {X 0,Y 432.46,Z 104.736,A -85,B 0,C 180,E1 -9372.196,E2 -9372.196} C_VEL
LIN {X 0,Y 432.431,Z 104.734,A -85,B 0,C 180,E1 -9376.039,E2 -9376.039} C_VEL
LIN {X 0,Y 432.388,Z 104.746,A -85,B 0,C 180,E1 -9379.485,E2 -9379.485} C_VEL
LIN {X 0,Y 432.32,Z 104.759,A -85,B 0,C 180,E1 -9382.964,E2 -9382.964} C_VEL
LIN {X 0,Y 432.365,Z 104.747,A -85,B 0,C 180,E1 -9386.032,E2 -9386.032} C_VEL
LIN {X 0,Y 432.344,Z 104.753,A -85,B 0,C 180,E1 -9389.187,E2 -9389.187} C_VEL
LIN {X 0,Y 432.324,Z 104.755,A -85,B 0,C 180,E1 -9392.443,E2 -9392.443} C_VEL
LIN {X 0,Y 432.345,Z 104.749,A -85,B 0,C 180,E1 -9395.632,E2 -9395.632} C_VEL
LIN {X 0,Y 432.338,Z 104.747,A -85,B 0,C 180,E1 -9398.714,E2 -9398.714} C_VEL
LIN {X 0,Y 432.334,Z 104.754,A -85,B 0,C 180,E1 -9401.797,E2 -9401.797} C_VEL
LIN {X 0,Y 432.334,Z 104.749,A -85,B 0,C 180,E1 -9404.347,E2 -9404.347} C_VEL
LIN {X 0,Y 432.321,Z 104.756,A -85,B 0,C 180,E1 -9407.016,E2 -9407.016} C_VEL
LIN {X 0,Y 432.342,Z 104.755,A -85,B 0,C 180,E1 -9409.819,E2 -9409.819} C_VEL
LIN {X 0,Y 432.307,Z 104.755,A -85,B 0,C 180,E1 -9413.022,E2 -9413.022} C_VEL
LIN {X 0,Y 432.36,Z 104.751,A -85,B 0,C 180,E1 -9415.996,E2 -9415.996} C_VEL
LIN {X 0,Y 432.348,Z 104.754,A -85,B 0,C 180,E1 -9419.49,E2 -9419.49} C_VEL
LIN {X 0,Y 432.369,Z 104.774,A -85,B 0,C 180,E1 -9420.414,E2 -9420.414} C_VEL
LIN {X 0,Y 435.476,Z 117.739,A -85,B 0,C 180,E1 -9423.135,E2 -9423.135} C_VEL
LIN {X 0,Y 436.781,Z 124.646,A -85,B 0,C 180,E1 -9424.518,E2 -9424.518} C_VEL
LIN {X 0,Y 435.617,Z 140.229,A -85,B 0,C 180,E1 -9427.322,E2 -9427.322} C_VEL
LIN {X 0,Y 435.684,Z 141.134,A -85,B 0,C 180,E1 -9427.386,E2 -9427.386} C_VEL
LIN {X 0,Y 440.24,Z 163.511,A -85,B 0,C 180,E1 -9428.047,E2 -9428.047} C_VEL
LIN {X 0,Y 440.885,Z 168.889,A -85,B 0,C 180,E1 -9428.178,E2 -9428.178} C_VEL
LIN {X 0,Y 439.342,Z 277.869,A -85,B 0,C 180,E1 -9430.005,E2 -9430.005} C_VEL
LIN {X 0,Y 438.785,Z 291.899,A -85,B 0,C 180,E1 -9430.406,E2 -9430.406} C_VEL
LIN {X 0,Y 438.055,Z 305.542,A -85,B 0,C 180,E1 -9430.981,E2 -9430.981} C_VEL
LIN {X 0,Y 437.204,Z 318.967,A -85,B 0,C 180,E1 -9431.744,E2 -9431.744} C_VEL
LIN {X 0,Y 436.269,Z 331.568,A -85,B 0,C 180,E1 -9432.661,E2 -9432.661} C_VEL
LIN {X 0,Y 435.266,Z 343.198,A -85,B 0,C 180,E1 -9433.707,E2 -9433.707} C_VEL
LIN {X 0,Y 434.443,Z 352.89,A -85,B 0,C 180,E1 -9434.759,E2 -9434.759} C_VEL
LIN {X 0,Y 433.541,Z 363.798,A -85,B 0,C 180,E1 -9436.19,E2 -9436.19} C_VEL
LIN {X 0,Y 432.873,Z 372.525,A -85,B 0,C 180,E1 -9437.577,E2 -9437.577} C_VEL
LIN {X 0,Y 432.166,Z 381.049,A -85,B 0,C 180,E1 -9439.221,E2 -9439.221} C_VEL
LIN {X 0,Y 431.766,Z 387.03,A -85,B 0,C 180,E1 -9440.632,E2 -9440.632} C_VEL
LIN {X 0,Y 431.419,Z 393.42,A -85,B 0,C 180,E1 -9442.512,E2 -9442.512} C_VEL
LIN {X 0,Y 431.265,Z 398.186,A -85,B 0,C 180,E1 -9444.389,E2 -9444.389} C_VEL
LIN {X 0,Y 431.156,Z 401.462,A -85,B 0,C 180,E1 -9446.261,E2 -9446.261} C_VEL
LIN {X 0,Y 431.198,Z 403.349,A -85,B 0,C 180,E1 -9448.132,E2 -9448.132} C_VEL
LIN {X 0,Y 431.143,Z 403.899,A -85,B 0,C 180,E1 -9450,E2 -9450} C_VEL
LIN {X 0,Y 431.199,Z 403.12,A -85,B 0,C 180,E1 -9451.868,E2 -9451.868} C_VEL
LIN {X 0,Y 431.157,Z 400.989,A -85,B 0,C 180,E1 -9453.738,E2 -9453.738} C_VEL
LIN {X 0,Y 431.243,Z 397.451,A -85,B 0,C 180,E1 -9455.611,E2 -9455.611} C_VEL
LIN {X 0,Y 431.408,Z 392.395,A -85,B 0,C 180,E1 -9457.488,E2 -9457.488} C_VEL
LIN {X 0,Y 431.715,Z 385.672,A -85,B 0,C 180,E1 -9459.369,E2 -9459.369} C_VEL
LIN {X 0,Y 432.167,Z 378.158,A -85,B 0,C 180,E1 -9461.016,E2 -9461.016} C_VEL
LIN {X 0,Y 432.759,Z 369.324,A -85,B 0,C 180,E1 -9462.584,E2 -9462.584} C_VEL
LIN {X 0,Y 433.292,Z 360.836,A -85,B 0,C 180,E1 -9463.842,E2 -9463.842} C_VEL
LIN {X 0,Y 434.037,Z 350.338,A -85,B 0,C 180,E1 -9465.135,E2 -9465.135} C_VEL
LIN {X 0,Y 434.931,Z 338.753,A -85,B 0,C 180,E1 -9466.305,E2 -9466.305} C_VEL
LIN {X 0,Y 435.828,Z 325.893,A -85,B 0,C 180,E1 -9467.357,E2 -9467.357} C_VEL
LIN {X 0,Y 436.673,Z 312.291,A -85,B 0,C 180,E1 -9468.232,E2 -9468.232} C_VEL
LIN {X 0,Y 437.358,Z 298.01,A -85,B 0,C 180,E1 -9468.929,E2 -9468.929} C_VEL
LIN {X 0,Y 437.967,Z 283.433,A -85,B 0,C 180,E1 -9469.419,E2 -9469.419} C_VEL
LIN {X 0,Y 438.287,Z 267.87,A -85,B 0,C 180,E1 -9469.739,E2 -9469.739} C_VEL
LIN {X 0,Y 439.451,Z 166.602,A -85,B 0,C 180,E1 -9471.402,E2 -9471.402} C_VEL
LIN {X 0,Y 434.929,Z 140.591,A -85,B 0,C 180,E1 -9472.067,E2 -9472.067} C_VEL
LIN {X 0,Y 436.024,Z 123.201,A -85,B 0,C 180,E1 -9475.12,E2 -9475.12} C_VEL
LIN {X 0,Y 435.548,Z 119.417,A -85,B 0,C 180,E1 -9475.828,E2 -9475.828} C_VEL
LIN {X 0,Y 432.773,Z 106.519,A -85,B 0,C 180,E1 -9478.356,E2 -9478.356} C_VEL
LIN {X 0,Y 432.367,Z 104.752,A -85,B 0,C 180,E1 -9478.743,E2 -9478.743} C_VEL
LIN {X 0,Y 432.321,Z 104.758,A -85,B 0,C 180,E1 -9481.346,E2 -9481.346} C_VEL
LIN {X 0,Y 432.339,Z 104.753,A -85,B 0,C 180,E1 -9484.677,E2 -9484.677} C_VEL
LIN {X 0,Y 432.336,Z 104.758,A -85,B 0,C 180,E1 -9488.15,E2 -9488.15} C_VEL
LIN {X 0,Y 432.332,Z 104.756,A -85,B 0,C 180,E1 -9491.602,E2 -9491.602} C_VEL
LIN {X 0,Y 432.337,Z 104.754,A -85,B 0,C 180,E1 -9494.347,E2 -9494.347} C_VEL
LIN {X 0,Y 432.366,Z 104.749,A -85,B 0,C 180,E1 -9497.009,E2 -9497.009} C_VEL
LIN {X 0,Y 432.334,Z 104.758,A -85,B 0,C 180,E1 -9499.82,E2 -9499.82} C_VEL
LIN {X 0,Y 432.305,Z 104.758,A -85,B 0,C 180,E1 -9503.022,E2 -9503.022} C_VEL
LIN {X 0,Y 432.358,Z 104.751,A -85,B 0,C 180,E1 -9505.996,E2 -9505.996} C_VEL
LIN {X 0,Y 432.346,Z 104.756,A -85,B 0,C 180,E1 -9509.49,E2 -9509.49} C_VEL
LIN {X 0,Y 432.39,Z 104.75,A -85,B 0,C 180,E1 -9512.928,E2 -9512.928} C_VEL
LIN {X 0,Y 432.37,Z 104.748,A -85,B 0,C 180,E1 -9516.023,E2 -9516.023} C_VEL
LIN {X 0,Y 432.349,Z 104.758,A -85,B 0,C 180,E1 -9519.046,E2 -9519.046} C_VEL
LIN {X 0,Y 432.376,Z 104.747,A -85,B 0,C 180,E1 -9522.011,E2 -9522.011} C_VEL
LIN {X 0,Y 432.395,Z 104.751,A -85,B 0,C 180,E1 -9524.927,E2 -9524.927} C_VEL
LIN {X 0,Y 432.458,Z 104.737,A -85,B 0,C 180,E1 -9527.804,E2 -9527.804} C_VEL
LIN {X 0,Y 432.491,Z 104.733,A -85,B 0,C 180,E1 -9531.59,E2 -9531.59} C_VEL
LIN {X 0,Y 432.593,Z 104.727,A -85,B 0,C 180,E1 -9534.406,E2 -9534.406} C_VEL
LIN {X 0,Y 432.602,Z 104.724,A -85,B 0,C 180,E1 -9538.138,E2 -9538.138} C_VEL
LIN {X 0,Y 432.731,Z 104.707,A -85,B 0,C 180,E1 -9540,E2 -9540} C_VEL
LIN {X 0,Y 432.591,Z 104.722,A -85,B 0,C 180,E1 -9542.794,E2 -9542.794} C_VEL
LIN {X 0,Y 432.584,Z 104.723,A -85,B 0,C 180,E1 -9545.594,E2 -9545.594} C_VEL
LIN {X 0,Y 432.482,Z 104.737,A -85,B 0,C 180,E1 -9548.41,E2 -9548.41} C_VEL
LIN {X 0,Y 432.459,Z 104.741,A -85,B 0,C 180,E1 -9552.197,E2 -9552.197} C_VEL
LIN {X 0,Y 432.429,Z 104.745,A -85,B 0,C 180,E1 -9556.039,E2 -9556.039} C_VEL
LIN {X 0,Y 432.385,Z 104.751,A -85,B 0,C 180,E1 -9559.485,E2 -9559.485} C_VEL
LIN {X 0,Y 432.317,Z 104.756,A -85,B 0,C 180,E1 -9562.965,E2 -9562.965} C_VEL
LIN {X 0,Y 432.36,Z 104.751,A -85,B 0,C 180,E1 -9566.033,E2 -9566.033} C_VEL
LIN {X 0,Y 432.342,Z 104.757,A -85,B 0,C 180,E1 -9569.188,E2 -9569.188} C_VEL
LIN {X 0,Y 432.322,Z 104.754,A -85,B 0,C 180,E1 -9572.443,E2 -9572.443} C_VEL
LIN {X 0,Y 432.343,Z 104.753,A -85,B 0,C 180,E1 -9575.632,E2 -9575.632} C_VEL
LIN {X 0,Y 432.339,Z 104.756,A -85,B 0,C 180,E1 -9578.715,E2 -9578.715} C_VEL
LIN {X 0,Y 432.333,Z 104.753,A -85,B 0,C 180,E1 -9581.797,E2 -9581.797} C_VEL
LIN {X 0,Y 432.334,Z 104.755,A -85,B 0,C 180,E1 -9584.348,E2 -9584.348} C_VEL
LIN {X 0,Y 432.317,Z 104.759,A -85,B 0,C 180,E1 -9587.017,E2 -9587.017} C_VEL
LIN {X 0,Y 432.332,Z 104.753,A -85,B 0,C 180,E1 -9589.821,E2 -9589.821} C_VEL
LIN {X 0,Y 432.306,Z 104.758,A -85,B 0,C 180,E1 -9593.022,E2 -9593.022} C_VEL
LIN {X 0,Y 432.36,Z 104.751,A -85,B 0,C 180,E1 -9595.997,E2 -9595.997} C_VEL
LIN {X 0,Y 432.348,Z 104.751,A -85,B 0,C 180,E1 -9599.49,E2 -9599.49} C_VEL
LIN {X 0,Y 432.349,Z 104.754,A -85,B 0,C 180,E1 -9601.875,E2 -9601.875} C_VEL
LIN {X 0,Y 432.379,Z 104.748,A -85,B 0,C 180,E1 -9605.539,E2 -9605.539} C_VEL
LIN {X 0,Y 432.353,Z 104.754,A -85,B 0,C 180,E1 -9609.046,E2 -9609.046} C_VEL
LIN {X 0,Y 432.405,Z 104.936,A -85,B 0,C 180,E1 -9610.258,E2 -9610.258} C_VEL
LIN {X 0,Y 434.749,Z 116.564,A -85,B 0,C 180,E1 -9612.769,E2 -9612.769} C_VEL
LIN {X 0,Y 435.349,Z 120.503,A -85,B 0,C 180,E1 -9613.59,E2 -9613.59} C_VEL
LIN {X 0,Y 435.192,Z 122.627,A -85,B 0,C 180,E1 -9614.006,E2 -9614.006} C_VEL
LIN {X 0,Y 439.733,Z 145.236,A -85,B 0,C 180,E1 -9614.621,E2 -9614.621} C_VEL
LIN {X 0,Y 438.449,Z 251.503,A -85,B 0,C 180,E1 -9616.365,E2 -9616.365} C_VEL
LIN {X 0,Y 437.791,Z 257.336,A -85,B 0,C 180,E1 -9616.448,E2 -9616.448} C_VEL
LIN {X 0,Y 434.902,Z 266.768,A -85,B 0,C 180,E1 -9616.573,E2 -9616.573} C_VEL
LIN {X 0,Y 431.82,Z 276.062,A -85,B 0,C 180,E1 -9616.774,E2 -9616.774} C_VEL
LIN {X 0,Y 430.891,Z 281.678,A -85,B 0,C 180,E1 -9616.982,E2 -9616.982} C_VEL
LIN {X 0,Y 430.243,Z 294.142,A -85,B 0,C 180,E1 -9617.62,E2 -9617.62} C_VEL
LIN {X 0,Y 429.436,Z 306.544,A -85,B 0,C 180,E1 -9618.435,E2 -9618.435} C_VEL
LIN {X 0,Y 428.544,Z 319.239,A -85,B 0,C 180,E1 -9619.488,E2 -9619.488} C_VEL
LIN {X 0,Y 427.655,Z 330.716,A -85,B 0,C 180,E1 -9620.664,E2 -9620.664} C_VEL
LIN {X 0,Y 426.962,Z 341.062,A -85,B 0,C 180,E1 -9621.957,E2 -9621.957} C_VEL
LIN {X 0,Y 426.134,Z 350.458,A -85,B 0,C 180,E1 -9623.371,E2 -9623.371} C_VEL
LIN {X 0,Y 425.402,Z 359.44,A -85,B 0,C 180,E1 -9625.024,E2 -9625.024} C_VEL
LIN {X 0,Y 424.848,Z 366.683,A -85,B 0,C 180,E1 -9626.681,E2 -9626.681} C_VEL
LIN {X 0,Y 424.461,Z 373.198,A -85,B 0,C 180,E1 -9628.577,E2 -9628.577} C_VEL
LIN {X 0,Y 424.272,Z 378.098,A -85,B 0,C 180,E1 -9630.475,E2 -9630.475} C_VEL
LIN {X 0,Y 424.174,Z 380.801,A -85,B 0,C 180,E1 -9631.899,E2 -9631.899} C_VEL
LIN {X 0,Y 424.08,Z 383.174,A -85,B 0,C 180,E1 -9633.801,E2 -9633.801} C_VEL
LIN {X 0,Y 424.114,Z 384.211,A -85,B 0,C 180,E1 -9635.706,E2 -9635.706} C_VEL
LIN {X 0,Y 424.079,Z 383.928,A -85,B 0,C 180,E1 -9637.619,E2 -9637.619} C_VEL
LIN {X 0,Y 424.056,Z 382.307,A -85,B 0,C 180,E1 -9639.54,E2 -9639.54} C_VEL
LIN {X 0,Y 424.291,Z 379.303,A -85,B 0,C 180,E1 -9641.465,E2 -9641.465} C_VEL
LIN {X 0,Y 424.567,Z 374.825,A -85,B 0,C 180,E1 -9643.4,E2 -9643.4} C_VEL
LIN {X 0,Y 424.858,Z 370.349,A -85,B 0,C 180,E1 -9644.857,E2 -9644.857} C_VEL
LIN {X 0,Y 425.454,Z 363.492,A -85,B 0,C 180,E1 -9646.645,E2 -9646.645} C_VEL
LIN {X 0,Y 426.115,Z 355.76,A -85,B 0,C 180,E1 -9648.263,E2 -9648.263} C_VEL
LIN {X 0,Y 426.904,Z 347.241,A -85,B 0,C 180,E1 -9649.724,E2 -9649.724} C_VEL
LIN {X 0,Y 427.886,Z 336.905,A -85,B 0,C 180,E1 -9651.183,E2 -9651.183} C_VEL
LIN {X 0,Y 428.8,Z 326.449,A -85,B 0,C 180,E1 -9652.4,E2 -9652.4} C_VEL
LIN {X 0,Y 429.838,Z 314.67,A -85,B 0,C 180,E1 -9653.52,E2 -9653.52} C_VEL
LIN {X 0,Y 430.76,Z 302.536,A -85,B 0,C 180,E1 -9654.457,E2 -9654.457} C_VEL
LIN {X 0,Y 431.69,Z 289.689,A -85,B 0,C 180,E1 -9655.235,E2 -9655.235} C_VEL
LIN {X 0,Y 432.346,Z 275.912,A -85,B 0,C 180,E1 -9655.872,E2 -9655.872} C_VEL
LIN {X 0,Y 432.878,Z 261.656,A -85,B 0,C 180,E1 -9656.325,E2 -9656.325} C_VEL
LIN {X 0,Y 433.331,Z 236.826,A -85,B 0,C 180,E1 -9656.782,E2 -9656.782} C_VEL
LIN {X 0,Y 434.575,Z 146.081,A -85,B 0,C 180,E1 -9658.318,E2 -9658.318} C_VEL
LIN {X 0,Y 430.057,Z 126.584,A -85,B 0,C 180,E1 -9658.944,E2 -9658.944} C_VEL
LIN {X 0,Y 428.951,Z 122.925,A -85,B 0,C 180,E1 -9659.094,E2 -9659.094} C_VEL
LIN {X 0,Y 426.879,Z 112.732,A -85,B 0,C 180,E1 -9661.406,E2 -9661.406} C_VEL
LIN {X 0,Y 425.285,Z 105.634,A -85,B 0,C 180,E1 -9663.118,E2 -9663.118} C_VEL
LIN {X 0,Y 425.257,Z 105.635,A -85,B 0,C 180,E1 -9666.509,E2 -9666.509} C_VEL
LIN {X 0,Y 425.245,Z 105.639,A -85,B 0,C 180,E1 -9669.034,E2 -9669.034} C_VEL
LIN {X 0,Y 425.256,Z 105.637,A -85,B 0,C 180,E1 -9672.655,E2 -9672.655} C_VEL
LIN {X 0,Y 425.284,Z 105.63,A -85,B 0,C 180,E1 -9675.283,E2 -9675.283} C_VEL
LIN {X 0,Y 425.249,Z 105.637,A -85,B 0,C 180,E1 -9678.618,E2 -9678.618} C_VEL
LIN {X 0,Y 425.277,Z 105.626,A -85,B 0,C 180,E1 -9681.099,E2 -9681.099} C_VEL
LIN {X 0,Y 425.295,Z 105.63,A -85,B 0,C 180,E1 -9684.663,E2 -9684.663} C_VEL
LIN {X 0,Y 425.265,Z 105.635,A -85,B 0,C 180,E1 -9688.073,E2 -9688.073} C_VEL
LIN {X 0,Y 425.306,Z 105.633,A -85,B 0,C 180,E1 -9691.366,E2 -9691.366} C_VEL
LIN {X 0,Y 425.26,Z 105.634,A -85,B 0,C 180,E1 -9694.552,E2 -9694.552} C_VEL
LIN {X 0,Y 425.292,Z 105.625,A -85,B 0,C 180,E1 -9697.73,E2 -9697.73} C_VEL
LIN {X 0,Y 425.362,Z 105.624,A -85,B 0,C 180,E1 -9700.704,E2 -9700.704} C_VEL
LIN {X 0,Y 425.389,Z 105.619,A -85,B 0,C 180,E1 -9703.688,E2 -9703.688} C_VEL
LIN {X 0,Y 425.413,Z 105.614,A -85,B 0,C 180,E1 -9707.598,E2 -9707.598} C_VEL
LIN {X 0,Y 425.409,Z 105.609,A -85,B 0,C 180,E1 -9711.449,E2 -9711.449} C_VEL
LIN {X 0,Y 425.54,Z 105.603,A -85,B 0,C 180,E1 -9714.313,E2 -9714.313} C_VEL
LIN {X 0,Y 425.573,Z 105.601,A -85,B 0,C 180,E1 -9718.107,E2 -9718.107} C_VEL
LIN {X 0,Y 425.7,Z 105.58,A -85,B 0,C 180,E1 -9720,E2 -9720} C_VEL
LIN {X 0,Y 425.538,Z 105.599,A -85,B 0,C 180,E1 -9722.84,E2 -9722.84} C_VEL
LIN {X 0,Y 425.533,Z 105.599,A -85,B 0,C 180,E1 -9725.687,E2 -9725.687} C_VEL
LIN {X 0,Y 425.409,Z 105.617,A -85,B 0,C 180,E1 -9728.551,E2 -9728.551} C_VEL
LIN {X 0,Y 425.413,Z 105.613,A -85,B 0,C 180,E1 -9732.402,E2 -9732.402} C_VEL
LIN {X 0,Y 425.389,Z 105.611,A -85,B 0,C 180,E1 -9736.312,E2 -9736.312} C_VEL
LIN {X 0,Y 425.329,Z 105.624,A -85,B 0,C 180,E1 -9739.636,E2 -9739.636} C_VEL
LIN {X 0,Y 425.307,Z 105.63,A -85,B 0,C 180,E1 -9743.365,E2 -9743.365} C_VEL
LIN {X 0,Y 425.348,Z 105.627,A -85,B 0,C 180,E1 -9746.844,E2 -9746.844} C_VEL
LIN {X 0,Y 425.292,Z 105.63,A -85,B 0,C 180,E1 -9749.719,E2 -9749.719} C_VEL
LIN {X 0,Y 425.283,Z 105.636,A -85,B 0,C 180,E1 -9753.048,E2 -9753.048} C_VEL
LIN {X 0,Y 425.283,Z 105.629,A -85,B 0,C 180,E1 -9755.929,E2 -9755.929} C_VEL
LIN {X 0,Y 425.281,Z 105.623,A -85,B 0,C 180,E1 -9759.041,E2 -9759.041} C_VEL
LIN {X 0,Y 425.29,Z 105.632,A -85,B 0,C 180,E1 -9761.958,E2 -9761.958} C_VEL
LIN {X 0,Y 425.285,Z 105.628,A -85,B 0,C 180,E1 -9765.283,E2 -9765.283} C_VEL
LIN {X 0,Y 425.276,Z 105.635,A -85,B 0,C 180,E1 -9768.621,E2 -9768.621} C_VEL
LIN {X 0,Y 425.313,Z 105.626,A -85,B 0,C 180,E1 -9771.103,E2 -9771.103} C_VEL
LIN {X 0,Y 425.3,Z 105.628,A -85,B 0,C 180,E1 -9774.664,E2 -9774.664} C_VEL
LIN {X 0,Y 425.266,Z 105.635,A -85,B 0,C 180,E1 -9778.073,E2 -9778.073} C_VEL
LIN {X 0,Y 425.336,Z 105.71,A -85,B 0,C 180,E1 -9780.045,E2 -9780.045} C_VEL
LIN {X 0,Y 428.571,Z 119.171,A -85,B 0,C 180,E1 -9782.931,E2 -9782.931} C_VEL
LIN {X 0,Y 429.953,Z 126.801,A -85,B 0,C 180,E1 -9784.482,E2 -9784.482} C_VEL
LIN {X 0,Y 428.842,Z 140.295,A -85,B 0,C 180,E1 -9786.949,E2 -9786.949} C_VEL
LIN {X 0,Y 433.749,Z 164.391,A -85,B 0,C 180,E1 -9787.685,E2 -9787.685} C_VEL
LIN {X 0,Y 434.386,Z 169.609,A -85,B 0,C 180,E1 -9787.815,E2 -9787.815} C_VEL
LIN {X 0,Y 432.769,Z 277.815,A -85,B 0,C 180,E1 -9789.658,E2 -9789.658} C_VEL
LIN {X 0,Y 432.159,Z 291.798,A -85,B 0,C 180,E1 -9790.062,E2 -9790.062} C_VEL
LIN {X 0,Y 431.366,Z 305.984,A -85,B 0,C 180,E1 -9790.674,E2 -9790.674} C_VEL
LIN {X 0,Y 430.456,Z 319.736,A -85,B 0,C 180,E1 -9791.48,E2 -9791.48} C_VEL
LIN {X 0,Y 429.5,Z 331.781,A -85,B 0,C 180,E1 -9792.379,E2 -9792.379} C_VEL
LIN {X 0,Y 428.454,Z 343.343,A -85,B 0,C 180,E1 -9793.441,E2 -9793.441} C_VEL
LIN {X 0,Y 427.569,Z 352.983,A -85,B 0,C 180,E1 -9794.508,E2 -9794.508} C_VEL
LIN {X 0,Y 426.609,Z 363.846,A -85,B 0,C 180,E1 -9795.961,E2 -9795.961} C_VEL
LIN {X 0,Y 425.879,Z 372.684,A -85,B 0,C 180,E1 -9797.397,E2 -9797.397} C_VEL
LIN {X 0,Y 425.141,Z 381.027,A -85,B 0,C 180,E1 -9799.041,E2 -9799.041} C_VEL
LIN {X 0,Y 424.726,Z 386.981,A -85,B 0,C 180,E1 -9800.475,E2 -9800.475} C_VEL
LIN {X 0,Y 424.344,Z 393.345,A -85,B 0,C 180,E1 -9802.386,E2 -9802.386} C_VEL
LIN {X 0,Y 424.175,Z 398.086,A -85,B 0,C 180,E1 -9804.295,E2 -9804.295} C_VEL
LIN {X 0,Y 424.166,Z 399.891,A -85,B 0,C 180,E1 -9805.248,E2 -9805.248} C_VEL
LIN {X 0,Y 424.09,Z 402.436,A -85,B 0,C 180,E1 -9807.15,E2 -9807.15} C_VEL
LIN {X 0,Y 424.067,Z 403.632,A -85,B 0,C 180,E1 -9809.05,E2 -9809.05} C_VEL
LIN {X 0,Y 424.067,Z 403.499,A -85,B 0,C 180,E1 -9810.949,E2 -9810.949} C_VEL
LIN {X 0,Y 424.118,Z 402.03,A -85,B 0,C 180,E1 -9812.849,E2 -9812.849} C_VEL
LIN {X 0,Y 424.16,Z 399.186,A -85,B 0,C 180,E1 -9814.752,E2 -9814.752} C_VEL
LIN {X 0,Y 424.222,Z 394.88,A -85,B 0,C 180,E1 -9816.659,E2 -9816.659} C_VEL
LIN {X 0,Y 424.457,Z 388.989,A -85,B 0,C 180,E1 -9818.57,E2 -9818.57} C_VEL
LIN {X 0,Y 424.799,Z 382.346,A -85,B 0,C 180,E1 -9820.244,E2 -9820.244} C_VEL
LIN {X 0,Y 425.428,Z 374.083,A -85,B 0,C 180,E1 -9821.917,E2 -9821.917} C_VEL
LIN {X 0,Y 425.965,Z 365.429,A -85,B 0,C 180,E1 -9823.355,E2 -9823.355} C_VEL
LIN {X 0,Y 426.806,Z 354.935,A -85,B 0,C 180,E1 -9824.787,E2 -9824.787} C_VEL
LIN {X 0,Y 427.564,Z 344.365,A -85,B 0,C 180,E1 -9825.981,E2 -9825.981} C_VEL
LIN {X 0,Y 428.459,Z 332.859,A -85,B 0,C 180,E1 -9827.05,E2 -9827.05} C_VEL
LIN {X 0,Y 429.402,Z 320.242,A -85,B 0,C 180,E1 -9827.994,E2 -9827.994} C_VEL
LIN {X 0,Y 430.158,Z 307.046,A -85,B 0,C 180,E1 -9828.772,E2 -9828.772} C_VEL
LIN {X 0,Y 430.808,Z 293.23,A -85,B 0,C 180,E1 -9829.383,E2 -9829.383} C_VEL
LIN {X 0,Y 431.359,Z 278.621,A -85,B 0,C 180,E1 -9829.821,E2 -9829.821} C_VEL
LIN {X 0,Y 432.849,Z 168.52,A -85,B 0,C 180,E1 -9831.676,E2 -9831.676} C_VEL
LIN {X 0,Y 428.026,Z 140.401,A -85,B 0,C 180,E1 -9832.41,E2 -9832.41} C_VEL
LIN {X 0,Y 429.094,Z 124.746,A -85,B 0,C 180,E1 -9835.204,E2 -9835.204} C_VEL
LIN {X 0,Y 428.473,Z 120.041,A -85,B 0,C 180,E1 -9836.102,E2 -9836.102} C_VEL
LIN {X 0,Y 425.332,Z 105.7,A -85,B 0,C 180,E1 -9838.978,E2 -9838.978} C_VEL
LIN {X 0,Y 425.281,Z 105.634,A -85,B 0,C 180,E1 -9842.563,E2 -9842.563} C_VEL
LIN {X 0,Y 425.299,Z 105.629,A -85,B 0,C 180,E1 -9845.336,E2 -9845.336} C_VEL
LIN {X 0,Y 425.293,Z 105.63,A -85,B 0,C 180,E1 -9849.043,E2 -9849.043} C_VEL
LIN {X 0,Y 425.274,Z 105.632,A -85,B 0,C 180,E1 -9852.653,E2 -9852.653} C_VEL
LIN {X 0,Y 425.334,Z 105.628,A -85,B 0,C 180,E1 -9856.054,E2 -9856.054} C_VEL
LIN {X 0,Y 425.3,Z 105.629,A -85,B 0,C 180,E1 -9858.625,E2 -9858.625} C_VEL
LIN {X 0,Y 425.296,Z 105.631,A -85,B 0,C 180,E1 -9861.101,E2 -9861.101} C_VEL
LIN {X 0,Y 425.298,Z 105.629,A -85,B 0,C 180,E1 -9864.664,E2 -9864.664} C_VEL
LIN {X 0,Y 425.264,Z 105.634,A -85,B 0,C 180,E1 -9868.073,E2 -9868.073} C_VEL
LIN {X 0,Y 425.33,Z 105.631,A -85,B 0,C 180,E1 -9871.368,E2 -9871.368} C_VEL
LIN {X 0,Y 425.294,Z 105.631,A -85,B 0,C 180,E1 -9874.555,E2 -9874.555} C_VEL
LIN {X 0,Y 425.286,Z 105.632,A -85,B 0,C 180,E1 -9877.661,E2 -9877.661} C_VEL
LIN {X 0,Y 425.361,Z 105.626,A -85,B 0,C 180,E1 -9880.704,E2 -9880.704} C_VEL
LIN {X 0,Y 425.387,Z 105.618,A -85,B 0,C 180,E1 -9883.688,E2 -9883.688} C_VEL
LIN {X 0,Y 425.411,Z 105.615,A -85,B 0,C 180,E1 -9887.598,E2 -9887.598} C_VEL
LIN {X 0,Y 425.441,Z 105.611,A -85,B 0,C 180,E1 -9891.45,E2 -9891.45} C_VEL
LIN {X 0,Y 425.55,Z 105.603,A -85,B 0,C 180,E1 -9894.313,E2 -9894.313} C_VEL
LIN {X 0,Y 425.572,Z 105.599,A -85,B 0,C 180,E1 -9898.107,E2 -9898.107} C_VEL
LIN {X 0,Y 425.7,Z 105.583,A -85,B 0,C 180,E1 -9900,E2 -9900} C_VEL
LIN {X 0,Y 425.545,Z 105.599,A -85,B 0,C 180,E1 -9902.84,E2 -9902.84} C_VEL
LIN {X 0,Y 425.496,Z 105.605,A -85,B 0,C 180,E1 -9906.531,E2 -9906.531} C_VEL
LIN {X 0,Y 425.4,Z 105.618,A -85,B 0,C 180,E1 -9909.51,E2 -9909.51} C_VEL
LIN {X 0,Y 425.393,Z 105.617,A -85,B 0,C 180,E1 -9912.904,E2 -9912.904} C_VEL
LIN {X 0,Y 425.36,Z 105.621,A -85,B 0,C 180,E1 -9916.605,E2 -9916.605} C_VEL
LIN {X 0,Y 425.327,Z 105.633,A -85,B 0,C 180,E1 -9919.636,E2 -9919.636} C_VEL
LIN {X 0,Y 425.304,Z 105.633,A -85,B 0,C 180,E1 -9923.366,E2 -9923.366} C_VEL
LIN {X 0,Y 425.346,Z 105.624,A -85,B 0,C 180,E1 -9926.844,E2 -9926.844} C_VEL
LIN {X 0,Y 425.29,Z 105.633,A -85,B 0,C 180,E1 -9929.72,E2 -9929.72} C_VEL
LIN {X 0,Y 425.281,Z 105.636,A -85,B 0,C 180,E1 -9933.048,E2 -9933.048} C_VEL
LIN {X 0,Y 425.281,Z 105.631,A -85,B 0,C 180,E1 -9935.929,E2 -9935.929} C_VEL
LIN {X 0,Y 425.283,Z 105.638,A -85,B 0,C 180,E1 -9939.041,E2 -9939.041} C_VEL
LIN {X 0,Y 425.29,Z 105.63,A -85,B 0,C 180,E1 -9941.959,E2 -9941.959} C_VEL
LIN {X 0,Y 425.285,Z 105.633,A -85,B 0,C 180,E1 -9945.283,E2 -9945.283} C_VEL
LIN {X 0,Y 425.268,Z 105.639,A -85,B 0,C 180,E1 -9948.621,E2 -9948.621} C_VEL
LIN {X 0,Y 425.292,Z 105.632,A -85,B 0,C 180,E1 -9951.101,E2 -9951.101} C_VEL
LIN {X 0,Y 425.3,Z 105.634,A -85,B 0,C 180,E1 -9954.664,E2 -9954.664} C_VEL
LIN {X 0,Y 425.267,Z 105.636,A -85,B 0,C 180,E1 -9958.074,E2 -9958.074} C_VEL
LIN {X 0,Y 425.315,Z 105.627,A -85,B 0,C 180,E1 -9961.367,E2 -9961.367} C_VEL
LIN {X 0,Y 425.272,Z 105.635,A -85,B 0,C 180,E1 -9964.553,E2 -9964.553} C_VEL
LIN {X 0,Y 425.286,Z 105.632,A -85,B 0,C 180,E1 -9966.634,E2 -9966.634} C_VEL
LIN {X 0,Y 425.347,Z 105.71,A -85,B 0,C 180,E1 -9969.973,E2 -9969.973} C_VEL
LIN {X 0,Y 427.623,Z 116.785,A -85,B 0,C 180,E1 -9972.409,E2 -9972.409} C_VEL
LIN {X 0,Y 428.382,Z 122.227,A -85,B 0,C 180,E1 -9973.561,E2 -9973.561} C_VEL
LIN {X 0,Y 428.356,Z 122.834,A -85,B 0,C 180,E1 -9973.682,E2 -9973.682} C_VEL
LIN {X 0,Y 433.043,Z 145.982,A -85,B 0,C 180,E1 -9974.317,E2 -9974.317} C_VEL
LIN {X 0,Y 431.563,Z 259.165,A -85,B 0,C 180,E1 -9976.222,E2 -9976.222} C_VEL
LIN {X 0,Y 431.158,Z 273.824,A -85,B 0,C 180,E1 -9976.659,E2 -9976.659} C_VEL
LIN {X 0,Y 430.891,Z 281.678,A -85,B 0,C 180,E1 -9976.982,E2 -9976.982} C_VEL
LIN {X 0,Y 429.927,Z 287.313,A -85,B 0,C 180,E1 -9977.218,E2 -9977.218} C_VEL
LIN {X 0,Y 426.684,Z 296.225,A -85,B 0,C 180,E1 -9977.603,E2 -9977.603} C_VEL
LIN {X 0,Y 423.403,Z 304.905,A -85,B 0,C 180,E1 -9978.066,E2 -9978.066} C_VEL
LIN {X 0,Y 422.405,Z 309.983,A -85,B 0,C 180,E1 -9978.426,E2 -9978.426} C_VEL
LIN {X 0,Y 421.547,Z 321.416,A -85,B 0,C 180,E1 -9979.433,E2 -9979.433} C_VEL
LIN {X 0,Y 420.57,Z 333.658,A -85,B 0,C 180,E1 -9980.768,E2 -9980.768} C_VEL
LIN {X 0,Y 419.817,Z 343.395,A -85,B 0,C 180,E1 -9982.062,E2 -9982.062} C_VEL
LIN {X 0,Y 419.025,Z 352.407,A -85,B 0,C 180,E1 -9983.5,E2 -9983.5} C_VEL
LIN {X 0,Y 418.203,Z 361.037,A -85,B 0,C 180,E1 -9985.18,E2 -9985.18} C_VEL
LIN {X 0,Y 417.795,Z 367.109,A -85,B 0,C 180,E1 -9986.625,E2 -9986.625} C_VEL
LIN {X 0,Y 417.392,Z 373.569,A -85,B 0,C 180,E1 -9988.553,E2 -9988.553} C_VEL
LIN {X 0,Y 417.171,Z 378.418,A -85,B 0,C 180,E1 -9990.483,E2 -9990.483} C_VEL
LIN {X 0,Y 417.099,Z 381.071,A -85,B 0,C 180,E1 -9991.931,E2 -9991.931} C_VEL
LIN {X 0,Y 416.993,Z 383.396,A -85,B 0,C 180,E1 -9993.866,E2 -9993.866} C_VEL
LIN {X 0,Y 417.036,Z 384.385,A -85,B 0,C 180,E1 -9995.803,E2 -9995.803} C_VEL
LIN {X 0,Y 416.979,Z 384.056,A -85,B 0,C 180,E1 -9997.749,E2 -9997.749} C_VEL
LIN {X 0,Y 416.974,Z 382.388,A -85,B 0,C 180,E1 -9999.704,E2 -9999.704} C_VEL
LIN {X 0,Y 417.24,Z 379.335,A -85,B 0,C 180,E1 -10001.662,E2 -10001.662} C_VEL
LIN {X 0,Y 417.529,Z 374.798,A -85,B 0,C 180,E1 -10003.63,E2 -10003.63} C_VEL
LIN {X 0,Y 417.872,Z 370.273,A -85,B 0,C 180,E1 -10005.111,E2 -10005.111} C_VEL
LIN {X 0,Y 418.446,Z 363.914,A -85,B 0,C 180,E1 -10006.794,E2 -10006.794} C_VEL
LIN {X 0,Y 419.085,Z 356.803,A -85,B 0,C 180,E1 -10008.327,E2 -10008.327} C_VEL
LIN {X 0,Y 419.916,Z 348.469,A -85,B 0,C 180,E1 -10009.811,E2 -10009.811} C_VEL
LIN {X 0,Y 420.933,Z 338.568,A -85,B 0,C 180,E1 -10011.268,E2 -10011.268} C_VEL
LIN {X 0,Y 421.867,Z 328.204,A -85,B 0,C 180,E1 -10012.53,E2 -10012.53} C_VEL
LIN {X 0,Y 423.051,Z 315.771,A -85,B 0,C 180,E1 -10013.761,E2 -10013.761} C_VEL
LIN {X 0,Y 424.036,Z 303.459,A -85,B 0,C 180,E1 -10014.74,E2 -10014.74} C_VEL
LIN {X 0,Y 425.017,Z 290.83,A -85,B 0,C 180,E1 -10015.529,E2 -10015.529} C_VEL
LIN {X 0,Y 425.722,Z 276.621,A -85,B 0,C 180,E1 -10016.206,E2 -10016.206} C_VEL
LIN {X 0,Y 426.324,Z 262.119,A -85,B 0,C 180,E1 -10016.678,E2 -10016.678} C_VEL
LIN {X 0,Y 426.742,Z 239.16,A -85,B 0,C 180,E1 -10017.114,E2 -10017.114} C_VEL
LIN {X 0,Y 428.111,Z 147.066,A -85,B 0,C 180,E1 -10018.694,E2 -10018.694} C_VEL
LIN {X 0,Y 423.568,Z 127.853,A -85,B 0,C 180,E1 -10019.333,E2 -10019.333} C_VEL
LIN {X 0,Y 421.852,Z 123.063,A -85,B 0,C 180,E1 -10019.555,E2 -10019.555} C_VEL
LIN {X 0,Y 419.207,Z 110.691,A -85,B 0,C 180,E1 -10022.444,E2 -10022.444} C_VEL
LIN {X 0,Y 418.246,Z 106.512,A -85,B 0,C 180,E1 -10023.459,E2 -10023.459} C_VEL
LIN {X 0,Y 418.239,Z 106.511,A -85,B 0,C 180,E1 -10026.236,E2 -10026.236} C_VEL
LIN {X 0,Y 418.194,Z 106.52,A -85,B 0,C 180,E1 -10029.688,E2 -10029.688} C_VEL
LIN {X 0,Y 418.207,Z 106.516,A -85,B 0,C 180,E1 -10032.317,E2 -10032.317} C_VEL
LIN {X 0,Y 418.235,Z 106.509,A -85,B 0,C 180,E1 -10035.108,E2 -10035.108} C_VEL
LIN {X 0,Y 418.22,Z 106.517,A -85,B 0,C 180,E1 -10037.764,E2 -10037.764} C_VEL
LIN {X 0,Y 418.235,Z 106.51,A -85,B 0,C 180,E1 -10041.556,E2 -10041.556} C_VEL
LIN {X 0,Y 418.251,Z 106.512,A -85,B 0,C 180,E1 -10045.158,E2 -10045.158} C_VEL
LIN {X 0,Y 418.245,Z 106.512,A -85,B 0,C 180,E1 -10047.472,E2 -10047.472} C_VEL
LIN {X 0,Y 418.263,Z 106.507,A -85,B 0,C 180,E1 -10050.897,E2 -10050.897} C_VEL
LIN {X 0,Y 418.229,Z 106.506,A -85,B 0,C 180,E1 -10054.093,E2 -10054.093} C_VEL
LIN {X 0,Y 418.228,Z 106.507,A -85,B 0,C 180,E1 -10057.263,E2 -10057.263} C_VEL
LIN {X 0,Y 418.284,Z 106.508,A -85,B 0,C 180,E1 -10060.364,E2 -10060.364} C_VEL
LIN {X 0,Y 418.317,Z 106.5,A -85,B 0,C 180,E1 -10063.404,E2 -10063.404} C_VEL
LIN {X 0,Y 418.348,Z 106.495,A -85,B 0,C 180,E1 -10066.999,E2 -10066.999} C_VEL
LIN {X 0,Y 418.339,Z 106.495,A -85,B 0,C 180,E1 -10070.328,E2 -10070.328} C_VEL
LIN {X 0,Y 418.46,Z 106.482,A -85,B 0,C 180,E1 -10073.248,E2 -10073.248} C_VEL
LIN {X 0,Y 418.333,Z 106.495,A -85,B 0,C 180,E1 -10075.181,E2 -10075.181} C_VEL
LIN {X 0,Y 418.542,Z 106.476,A -85,B 0,C 180,E1 -10078.075,E2 -10078.075} C_VEL
LIN {X 0,Y 418.67,Z 106.456,A -85,B 0,C 180,E1 -10080,E2 -10080} C_VEL
LIN {X 0,Y 418.494,Z 106.477,A -85,B 0,C 180,E1 -10082.888,E2 -10082.888} C_VEL
LIN {X 0,Y 418.49,Z 106.475,A -85,B 0,C 180,E1 -10085.783,E2 -10085.783} C_VEL
LIN {X 0,Y 418.378,Z 106.492,A -85,B 0,C 180,E1 -10088.695,E2 -10088.695} C_VEL
LIN {X 0,Y 418.315,Z 106.498,A -85,B 0,C 180,E1 -10091.631,E2 -10091.631} C_VEL
LIN {X 0,Y 418.303,Z 106.501,A -85,B 0,C 180,E1 -10094.597,E2 -10094.597} C_VEL
LIN {X 0,Y 418.288,Z 106.506,A -85,B 0,C 180,E1 -10097.604,E2 -10097.604} C_VEL
LIN {X 0,Y 418.251,Z 106.504,A -85,B 0,C 180,E1 -10100.663,E2 -10100.663} C_VEL
LIN {X 0,Y 418.289,Z 106.501,A -85,B 0,C 180,E1 -10103.781,E2 -10103.781} C_VEL
LIN {X 0,Y 418.311,Z 106.504,A -85,B 0,C 180,E1 -10107.07,E2 -10107.07} C_VEL
LIN {X 0,Y 418.245,Z 106.509,A -85,B 0,C 180,E1 -10110.272,E2 -10110.272} C_VEL
LIN {X 0,Y 418.249,Z 106.509,A -85,B 0,C 180,E1 -10113.677,E2 -10113.677} C_VEL
LIN {X 0,Y 418.24,Z 106.511,A -85,B 0,C 180,E1 -10117.224,E2 -10117.224} C_VEL
LIN {X 0,Y 418.244,Z 106.497,A -85,B 0,C 180,E1 -10119.683,E2 -10119.683} C_VEL
LIN {X 0,Y 418.23,Z 106.516,A -85,B 0,C 180,E1 -10122.321,E2 -10122.321} C_VEL
LIN {X 0,Y 418.236,Z 106.506,A -85,B 0,C 180,E1 -10125.109,E2 -10125.109} C_VEL
LIN {X 0,Y 418.241,Z 106.512,A -85,B 0,C 180,E1 -10127.767,E2 -10127.767} C_VEL
LIN {X 0,Y 418.259,Z 106.507,A -85,B 0,C 180,E1 -10130.618,E2 -10130.618} C_VEL
LIN {X 0,Y 418.244,Z 106.509,A -85,B 0,C 180,E1 -10133.976,E2 -10133.976} C_VEL
LIN {X 0,Y 418.258,Z 106.5,A -85,B 0,C 180,E1 -10137.156,E2 -10137.156} C_VEL
LIN {X 0,Y 418.298,Z 106.693,A -85,B 0,C 180,E1 -10139.671,E2 -10139.671} C_VEL
LIN {X 0,Y 421.322,Z 119.15,A -85,B 0,C 180,E1 -10142.408,E2 -10142.408} C_VEL
LIN {X 0,Y 422.946,Z 126.985,A -85,B 0,C 180,E1 -10144.053,E2 -10144.053} C_VEL
LIN {X 0,Y 422.839,Z 131.528,A -85,B 0,C 180,E1 -10144.923,E2 -10144.923} C_VEL
LIN {X 0,Y 422.102,Z 140.117,A -85,B 0,C 180,E1 -10146.517,E2 -10146.517} C_VEL
LIN {X 0,Y 427.424,Z 166.451,A -85,B 0,C 180,E1 -10147.342,E2 -10147.342} C_VEL
LIN {X 0,Y 427.931,Z 171.081,A -85,B 0,C 180,E1 -10147.456,E2 -10147.456} C_VEL
LIN {X 0,Y 426.199,Z 277.797,A -85,B 0,C 180,E1 -10149.298,E2 -10149.298} C_VEL
LIN {X 0,Y 425.572,Z 291.718,A -85,B 0,C 180,E1 -10149.708,E2 -10149.708} C_VEL
LIN {X 0,Y 424.752,Z 305.32,A -85,B 0,C 180,E1 -10150.298,E2 -10150.298} C_VEL
LIN {X 0,Y 423.831,Z 318.935,A -85,B 0,C 180,E1 -10151.1,E2 -10151.1} C_VEL
LIN {X 0,Y 422.749,Z 332.006,A -85,B 0,C 180,E1 -10152.088,E2 -10152.088} C_VEL
LIN {X 0,Y 421.659,Z 343.499,A -85,B 0,C 180,E1 -10153.166,E2 -10153.166} C_VEL
LIN {X 0,Y 420.545,Z 355.029,A -85,B 0,C 180,E1 -10154.491,E2 -10154.491} C_VEL
LIN {X 0,Y 419.555,Z 365.36,A -85,B 0,C 180,E1 -10155.943,E2 -10155.943} C_VEL
LIN {X 0,Y 418.809,Z 373.901,A -85,B 0,C 180,E1 -10157.399,E2 -10157.399} C_VEL
LIN {X 0,Y 418.065,Z 382.09,A -85,B 0,C 180,E1 -10159.098,E2 -10159.098} C_VEL
LIN {X 0,Y 417.553,Z 388.699,A -85,B 0,C 180,E1 -10160.799,E2 -10160.799} C_VEL
LIN {X 0,Y 417.242,Z 394.579,A -85,B 0,C 180,E1 -10162.742,E2 -10162.742} C_VEL
LIN {X 0,Y 417.091,Z 397.987,A -85,B 0,C 180,E1 -10164.197,E2 -10164.197} C_VEL
LIN {X 0,Y 416.985,Z 401.208,A -85,B 0,C 180,E1 -10166.134,E2 -10166.134} C_VEL
LIN {X 0,Y 417.049,Z 403.054,A -85,B 0,C 180,E1 -10168.068,E2 -10168.068} C_VEL
LIN {X 0,Y 416.982,Z 403.564,A -85,B 0,C 180,E1 -10170,E2 -10170} C_VEL
LIN {X 0,Y 417.052,Z 402.746,A -85,B 0,C 180,E1 -10171.931,E2 -10171.931} C_VEL
LIN {X 0,Y 416.985,Z 400.573,A -85,B 0,C 180,E1 -10173.865,E2 -10173.865} C_VEL
LIN {X 0,Y 417.065,Z 398.966,A -85,B 0,C 180,E1 -10174.833,E2 -10174.833} C_VEL
LIN {X 0,Y 417.153,Z 394.638,A -85,B 0,C 180,E1 -10176.773,E2 -10176.773} C_VEL
LIN {X 0,Y 417.406,Z 388.722,A -85,B 0,C 180,E1 -10178.716,E2 -10178.716} C_VEL
LIN {X 0,Y 417.773,Z 382.05,A -85,B 0,C 180,E1 -10180.419,E2 -10180.419} C_VEL
LIN {X 0,Y 418.39,Z 373.739,A -85,B 0,C 180,E1 -10182.12,E2 -10182.12} C_VEL
LIN {X 0,Y 418.994,Z 365.048,A -85,B 0,C 180,E1 -10183.581,E2 -10183.581} C_VEL
LIN {X 0,Y 419.867,Z 354.508,A -85,B 0,C 180,E1 -10185.037,E2 -10185.037} C_VEL
LIN {X 0,Y 420.756,Z 342.699,A -85,B 0,C 180,E1 -10186.371,E2 -10186.371} C_VEL
LIN {X 0,Y 421.727,Z 330.871,A -85,B 0,C 180,E1 -10187.455,E2 -10187.455} C_VEL
LIN {X 0,Y 422.693,Z 317.812,A -85,B 0,C 180,E1 -10188.415,E2 -10188.415} C_VEL
LIN {X 0,Y 423.494,Z 303.737,A -85,B 0,C 180,E1 -10189.215,E2 -10189.215} C_VEL
LIN {X 0,Y 424.223,Z 289.689,A -85,B 0,C 180,E1 -10189.79,E2 -10189.79} C_VEL
LIN {X 0,Y 424.695,Z 275.492,A -85,B 0,C 180,E1 -10190.177,E2 -10190.177} C_VEL
LIN {X 0,Y 426.091,Z 168.456,A -85,B 0,C 180,E1 -10192,E2 -10192} C_VEL
LIN {X 0,Y 421.197,Z 140.277,A -85,B 0,C 180,E1 -10192.75,E2 -10192.75} C_VEL
LIN {X 0,Y 422.191,Z 125.789,A -85,B 0,C 180,E1 -10195.381,E2 -10195.381} C_VEL
LIN {X 0,Y 420.966,Z 118.635,A -85,B 0,C 180,E1 -10196.792,E2 -10196.792} C_VEL
LIN {X 0,Y 418.25,Z 106.512,A -85,B 0,C 180,E1 -10199.301,E2 -10199.301} C_VEL
LIN {X 0,Y 418.257,Z 106.507,A -85,B 0,C 180,E1 -10202.844,E2 -10202.844} C_VEL
LIN {X 0,Y 418.245,Z 106.513,A -85,B 0,C 180,E1 -10206.238,E2 -10206.238} C_VEL
LIN {X 0,Y 418.248,Z 106.511,A -85,B 0,C 180,E1 -10209.682,E2 -10209.682} C_VEL
LIN {X 0,Y 418.229,Z 106.512,A -85,B 0,C 180,E1 -10212.321,E2 -10212.321} C_VEL
LIN {X 0,Y 418.259,Z 106.507,A -85,B 0,C 180,E1 -10215.112,E2 -10215.112} C_VEL
LIN {X 0,Y 418.29,Z 106.508,A -85,B 0,C 180,E1 -10217.773,E2 -10217.773} C_VEL
LIN {X 0,Y 418.247,Z 106.515,A -85,B 0,C 180,E1 -10221.558,E2 -10221.558} C_VEL
LIN {X 0,Y 418.258,Z 106.51,A -85,B 0,C 180,E1 -10225.159,E2 -10225.159} C_VEL
LIN {X 0,Y 418.244,Z 106.514,A -85,B 0,C 180,E1 -10227.472,E2 -10227.472} C_VEL
LIN {X 0,Y 418.267,Z 106.508,A -85,B 0,C 180,E1 -10230.895,E2 -10230.895} C_VEL
LIN {X 0,Y 418.269,Z 106.505,A -85,B 0,C 180,E1 -10234.096,E2 -10234.096} C_VEL
LIN {X 0,Y 418.237,Z 106.513,A -85,B 0,C 180,E1 -10237.264,E2 -10237.264} C_VEL
LIN {X 0,Y 418.282,Z 106.504,A -85,B 0,C 180,E1 -10240.364,E2 -10240.364} C_VEL
LIN {X 0,Y 418.316,Z 106.5,A -85,B 0,C 180,E1 -10243.405,E2 -10243.405} C_VEL
LIN {X 0,Y 418.345,Z 106.499,A -85,B 0,C 180,E1 -10246.999,E2 -10246.999} C_VEL
LIN {X 0,Y 418.34,Z 106.499,A -85,B 0,C 180,E1 -10250.329,E2 -10250.329} C_VEL
LIN {X 0,Y 418.487,Z 106.478,A -85,B 0,C 180,E1 -10253.249,E2 -10253.249} C_VEL
LIN {X 0,Y 418.337,Z 106.497,A -85,B 0,C 180,E1 -10255.182,E2 -10255.182} C_VEL
LIN {X 0,Y 418.541,Z 106.474,A -85,B 0,C 180,E1 -10258.076,E2 -10258.076} C_VEL
LIN {X 0,Y 418.67,Z 106.458,A -85,B 0,C 180,E1 -10260,E2 -10260} C_VEL
LIN {X 0,Y 418.5,Z 106.477,A -85,B 0,C 180,E1 -10262.888,E2 -10262.888} C_VEL
LIN {X 0,Y 418.457,Z 106.481,A -85,B 0,C 180,E1 -10266.53,E2 -10266.53} C_VEL
LIN {X 0,Y 418.34,Z 106.499,A -85,B 0,C 180,E1 -10269.672,E2 -10269.672} C_VEL
LIN {X 0,Y 418.346,Z 106.495,A -85,B 0,C 180,E1 -10273.001,E2 -10273.001} C_VEL
LIN {X 0,Y 418.312,Z 106.499,A -85,B 0,C 180,E1 -10276.735,E2 -10276.735} C_VEL
LIN {X 0,Y 418.27,Z 106.51,A -85,B 0,C 180,E1 -10279.79,E2 -10279.79} C_VEL
LIN {X 0,Y 418.237,Z 106.509,A -85,B 0,C 180,E1 -10282.736,E2 -10282.736} C_VEL
LIN {X 0,Y 418.268,Z 106.507,A -85,B 0,C 180,E1 -10285.905,E2 -10285.905} C_VEL
LIN {X 0,Y 418.264,Z 106.51,A -85,B 0,C 180,E1 -10289.162,E2 -10289.162} C_VEL
LIN {X 0,Y 418.257,Z 106.509,A -85,B 0,C 180,E1 -10292.844,E2 -10292.844} C_VEL
LIN {X 0,Y 418.244,Z 106.508,A -85,B 0,C 180,E1 -10296.238,E2 -10296.238} C_VEL
LIN {X 0,Y 418.245,Z 106.508,A -85,B 0,C 180,E1 -10299.683,E2 -10299.683} C_VEL
LIN {X 0,Y 418.23,Z 106.511,A -85,B 0,C 180,E1 -10302.321,E2 -10302.321} C_VEL
LIN {X 0,Y 418.236,Z 106.512,A -85,B 0,C 180,E1 -10305.109,E2 -10305.109} C_VEL
LIN {X 0,Y 418.235,Z 106.509,A -85,B 0,C 180,E1 -10307.766,E2 -10307.766} C_VEL
LIN {X 0,Y 418.242,Z 106.515,A -85,B 0,C 180,E1 -10310.622,E2 -10310.622} C_VEL
LIN {X 0,Y 418.243,Z 106.509,A -85,B 0,C 180,E1 -10313.976,E2 -10313.976} C_VEL
LIN {X 0,Y 418.259,Z 106.506,A -85,B 0,C 180,E1 -10317.156,E2 -10317.156} C_VEL
LIN {X 0,Y 418.262,Z 106.507,A -85,B 0,C 180,E1 -10320.838,E2 -10320.838} C_VEL
LIN {X 0,Y 418.237,Z 106.515,A -85,B 0,C 180,E1 -10324.094,E2 -10324.094} C_VEL
LIN {X 0,Y 418.234,Z 106.509,A -85,B 0,C 180,E1 -10327.264,E2 -10327.264} C_VEL
LIN {X 0,Y 418.306,Z 106.628,A -85,B 0,C 180,E1 -10329.707,E2 -10329.707} C_VEL
LIN {X 0,Y 420.651,Z 117.924,A -85,B 0,C 180,E1 -10332.238,E2 -10332.238} C_VEL
LIN {X 0,Y 421.462,Z 122.976,A -85,B 0,C 180,E1 -10333.33,E2 -10333.33} C_VEL
LIN {X 0,Y 426.356,Z 147.089,A -85,B 0,C 180,E1 -10334.011,E2 -10334.011} C_VEL
LIN {X 0,Y 424.821,Z 259.708,A -85,B 0,C 180,E1 -10335.938,E2 -10335.938} C_VEL
LIN {X 0,Y 424.408,Z 274.215,A -85,B 0,C 180,E1 -10336.382,E2 -10336.382} C_VEL
LIN {X 0,Y 423.749,Z 288.094,A -85,B 0,C 180,E1 -10337.001,E2 -10337.001} C_VEL
LIN {X 0,Y 422.954,Z 301.01,A -85,B 0,C 180,E1 -10337.769,E2 -10337.769} C_VEL
LIN {X 0,Y 422.405,Z 309.983,A -85,B 0,C 180,E1 -10338.426,E2 -10338.426} C_VEL
LIN {X 0,Y 421.38,Z 315.047,A -85,B 0,C 180,E1 -10338.818,E2 -10338.818} C_VEL
LIN {X 0,Y 417.953,Z 323.077,A -85,B 0,C 180,E1 -10339.464,E2 -10339.464} C_VEL
LIN {X 0,Y 414.537,Z 330.742,A -85,B 0,C 180,E1 -10340.194,E2 -10340.194} C_VEL
LIN {X 0,Y 413.54,Z 335.173,A -85,B 0,C 180,E1 -10340.711,E2 -10340.711} C_VEL
LIN {X 0,Y 412.811,Z 344.025,A -85,B 0,C 180,E1 -10341.926,E2 -10341.926} C_VEL
LIN {X 0,Y 412.008,Z 352.957,A -85,B 0,C 180,E1 -10343.388,E2 -10343.388} C_VEL
LIN {X 0,Y 411.164,Z 361.52,A -85,B 0,C 180,E1 -10345.097,E2 -10345.097} C_VEL
LIN {X 0,Y 410.743,Z 367.532,A -85,B 0,C 180,E1 -10346.567,E2 -10346.567} C_VEL
LIN {X 0,Y 410.326,Z 373.938,A -85,B 0,C 180,E1 -10348.528,E2 -10348.528} C_VEL
LIN {X 0,Y 410.075,Z 378.735,A -85,B 0,C 180,E1 -10350.491,E2 -10350.491} C_VEL
LIN {X 0,Y 410.025,Z 381.338,A -85,B 0,C 180,E1 -10351.965,E2 -10351.965} C_VEL
LIN {X 0,Y 409.908,Z 383.617,A -85,B 0,C 180,E1 -10353.933,E2 -10353.933} C_VEL
LIN {X 0,Y 409.958,Z 384.56,A -85,B 0,C 180,E1 -10355.904,E2 -10355.904} C_VEL
LIN {X 0,Y 409.876,Z 384.184,A -85,B 0,C 180,E1 -10357.884,E2 -10357.884} C_VEL
